LIN {X 0,Y 573.263,Z 379.078,A -85,B 0,C 180,E1 -2328.745,E2 -2328.745} C_VEL
LIN {X 0,Y 573.288,Z 379.077,A -85,B 0,C 180,E1 -2331.54,E2 -2331.54} C_VEL
LIN {X 0,Y 573.291,Z 379.075,A -85,B 0,C 180,E1 -2334.372,E2 -2334.372} C_VEL
LIN {X 0,Y 573.302,Z 379.074,A -85,B 0,C 180,E1 -2337.892,E2 -2337.892} C_VEL
LIN {X 0,Y 573.331,Z 379.07,A -85,B 0,C 180,E1 -2340.702,E2 -2340.702} C_VEL
LIN {X 0,Y 573.236,Z 379.084,A -85,B 0,C 180,E1 -2343.514,E2 -2343.514} C_VEL
LIN {X 0,Y 573.289,Z 379.075,A -85,B 0,C 180,E1 -2345.628,E2 -2345.628} C_VEL
LIN {X 0,Y 573.288,Z 379.078,A -85,B 0,C 180,E1 -2348.459,E2 -2348.459} C_VEL
LIN {X 0,Y 573.272,Z 379.077,A -85,B 0,C 180,E1 -2351.312,E2 -2351.312} C_VEL
LIN {X 0,Y 573.281,Z 379.079,A -85,B 0,C 180,E1 -2354.424,E2 -2354.424} C_VEL
LIN {X 0,Y 573.26,Z 379.079,A -85,B 0,C 180,E1 -2357.112,E2 -2357.112} C_VEL
LIN {X 0,Y 573.244,Z 379.081,A -85,B 0,C 180,E1 -2360.077,E2 -2360.077} C_VEL
LIN {X 0,Y 573.235,Z 379.082,A -85,B 0,C 180,E1 -2362.338,E2 -2362.338} C_VEL
LIN {X 0,Y 573.25,Z 379.079,A -85,B 0,C 180,E1 -2364.384,E2 -2364.384} C_VEL
LIN {X 0,Y 572.623,Z 379.16,A -85,B 0,C 180,E1 -2364.97,E2 -2364.97} C_VEL
LIN {X 0,Y 569.781,Z 379.516,A -85,B 0,C 180,E1 -2365.922,E2 -2365.922} C_VEL
LIN {X 0,Y 567.349,Z 379.82,A -85,B 0,C 180,E1 -2366.687,E2 -2366.687} C_VEL
LIN {X 0,Y 566.293,Z 379.949,A -85,B 0,C 180,E1 -2367.278,E2 -2367.278} C_VEL
LIN {X 0,Y 566.203,Z 379.958,A -85,B 0,C 180,E1 -2367.478,E2 -2367.478} C_VEL
LIN {X 0,Y 566.201,Z 379.96,A -85,B 0,C 180,E1 -2369.769,E2 -2369.769} C_VEL
LIN {X 0,Y 566.206,Z 379.959,A -85,B 0,C 180,E1 -2372.43,E2 -2372.43} C_VEL
LIN {X 0,Y 566.202,Z 379.958,A -85,B 0,C 180,E1 -2374.993,E2 -2374.993} C_VEL
LIN {X 0,Y 566.198,Z 379.957,A -85,B 0,C 180,E1 -2377.461,E2 -2377.461} C_VEL
LIN {X 0,Y 566.207,Z 379.957,A -85,B 0,C 180,E1 -2380.199,E2 -2380.199} C_VEL
LIN {X 0,Y 566.203,Z 379.96,A -85,B 0,C 180,E1 -2383.054,E2 -2383.054} C_VEL
LIN {X 0,Y 566.195,Z 379.958,A -85,B 0,C 180,E1 -2386.049,E2 -2386.049} C_VEL
LIN {X 0,Y 566.212,Z 379.959,A -85,B 0,C 180,E1 -2388.864,E2 -2388.864} C_VEL
LIN {X 0,Y 566.184,Z 379.96,A -85,B 0,C 180,E1 -2391.637,E2 -2391.637} C_VEL
LIN {X 0,Y 566.198,Z 379.958,A -85,B 0,C 180,E1 -2394.31,E2 -2394.31} C_VEL
LIN {X 0,Y 566.222,Z 379.955,A -85,B 0,C 180,E1 -2396.898,E2 -2396.898} C_VEL
LIN {X 0,Y 566.182,Z 379.961,A -85,B 0,C 180,E1 -2399.407,E2 -2399.407} C_VEL
LIN {X 0,Y 566.195,Z 379.959,A -85,B 0,C 180,E1 -2401.856,E2 -2401.856} C_VEL
LIN {X 0,Y 566.218,Z 379.957,A -85,B 0,C 180,E1 -2404.251,E2 -2404.251} C_VEL
LIN {X 0,Y 566.176,Z 379.963,A -85,B 0,C 180,E1 -2406.718,E2 -2406.718} C_VEL
LIN {X 0,Y 566.215,Z 379.956,A -85,B 0,C 180,E1 -2409.663,E2 -2409.663} C_VEL
LIN {X 0,Y 566.202,Z 379.96,A -85,B 0,C 180,E1 -2412.668,E2 -2412.668} C_VEL
LIN {X 0,Y 566.237,Z 379.953,A -85,B 0,C 180,E1 -2415.627,E2 -2415.627} C_VEL
LIN {X 0,Y 566.238,Z 379.956,A -85,B 0,C 180,E1 -2418.675,E2 -2418.675} C_VEL
LIN {X 0,Y 566.23,Z 379.955,A -85,B 0,C 180,E1 -2421.434,E2 -2421.434} C_VEL
LIN {X 0,Y 566.266,Z 379.95,A -85,B 0,C 180,E1 -2424.302,E2 -2424.302} C_VEL
LIN {X 0,Y 566.287,Z 379.947,A -85,B 0,C 180,E1 -2427.866,E2 -2427.866} C_VEL
LIN {X 0,Y 566.306,Z 379.947,A -85,B 0,C 180,E1 -2430.711,E2 -2430.711} C_VEL
LIN {X 0,Y 566.27,Z 379.95,A -85,B 0,C 180,E1 -2432.845,E2 -2432.845} C_VEL
LIN {X 0,Y 566.26,Z 379.952,A -85,B 0,C 180,E1 -2435.698,E2 -2435.698} C_VEL
LIN {X 0,Y 566.14,Z 379.968,A -85,B 0,C 180,E1 -2437.848,E2 -2437.848} C_VEL
LIN {X 0,Y 566.113,Z 380.449,A -85,B 0,C 180,E1 -2438.567,E2 -2438.567} C_VEL
LIN {X 0,Y 566.106,Z 384.738,A -85,B 0,C 180,E1 -2441.457,E2 -2441.457} C_VEL
LIN {X 0,Y 566.047,Z 389.206,A -85,B 0,C 180,E1 -2444.432,E2 -2444.432} C_VEL
LIN {X 0,Y 565.989,Z 393.668,A -85,B 0,C 180,E1 -2447.338,E2 -2447.338} C_VEL
LIN {X 0,Y 565.926,Z 397.067,A -85,B 0,C 180,E1 -2449.59,E2 -2449.59} C_VEL
LIN {X 0,Y 565.882,Z 401.918,A -85,B 0,C 180,E1 -2452.644,E2 -2452.644} C_VEL
LIN {X 0,Y 565.901,Z 405.761,A -85,B 0,C 180,E1 -2454.976,E2 -2454.976} C_VEL
LIN {X 0,Y 565.844,Z 409.742,A -85,B 0,C 180,E1 -2457.358,E2 -2457.358} C_VEL
LIN {X 0,Y 565.846,Z 414.922,A -85,B 0,C 180,E1 -2460.419,E2 -2460.419} C_VEL
LIN {X 0,Y 566.897,Z 422.356,A -85,B 0,C 180,E1 -2460.606,E2 -2460.606} C_VEL
LIN {X 0,Y 566.779,Z 435.719,A -85,B 0,C 180,E1 -2461.011,E2 -2461.011} C_VEL
LIN {X 0,Y 566.587,Z 448.306,A -85,B 0,C 180,E1 -2461.553,E2 -2461.553} C_VEL
LIN {X 0,Y 566.394,Z 460.453,A -85,B 0,C 180,E1 -2462.246,E2 -2462.246} C_VEL
LIN {X 0,Y 566.362,Z 470.852,A -85,B 0,C 180,E1 -2462.996,E2 -2462.996} C_VEL
LIN {X 0,Y 566.23,Z 480.115,A -85,B 0,C 180,E1 -2463.816,E2 -2463.816} C_VEL
LIN {X 0,Y 566.105,Z 489.376,A -85,B 0,C 180,E1 -2464.825,E2 -2464.825} C_VEL
LIN {X 0,Y 566.04,Z 497.674,A -85,B 0,C 180,E1 -2465.943,E2 -2465.943} C_VEL
LIN {X 0,Y 565.959,Z 503.812,A -85,B 0,C 180,E1 -2466.975,E2 -2466.975} C_VEL
LIN {X 0,Y 565.916,Z 508.408,A -85,B 0,C 180,E1 -2467.932,E2 -2467.932} C_VEL
LIN {X 0,Y 565.92,Z 512.057,A -85,B 0,C 180,E1 -2468.881,E2 -2468.881} C_VEL
LIN {X 0,Y 565.882,Z 515.874,A -85,B 0,C 180,E1 -2470.226,E2 -2470.226} C_VEL
LIN {X 0,Y 565.856,Z 517.602,A -85,B 0,C 180,E1 -2471.167,E2 -2471.167} C_VEL
LIN {X 0,Y 565.862,Z 518.643,A -85,B 0,C 180,E1 -2472.119,E2 -2472.119} C_VEL
LIN {X 0,Y 565.848,Z 518.997,A -85,B 0,C 180,E1 -2473.087,E2 -2473.087} C_VEL
LIN {X 0,Y 565.861,Z 518.578,A -85,B 0,C 180,E1 -2474.068,E2 -2474.068} C_VEL
LIN {X 0,Y 565.88,Z 517.38,A -85,B 0,C 180,E1 -2475.065,E2 -2475.065} C_VEL
LIN {X 0,Y 565.871,Z 515.34,A -85,B 0,C 180,E1 -2476.082,E2 -2476.082} C_VEL
LIN {X 0,Y 565.902,Z 512.383,A -85,B 0,C 180,E1 -2477.115,E2 -2477.115} C_VEL
LIN {X 0,Y 565.944,Z 508.372,A -85,B 0,C 180,E1 -2478.166,E2 -2478.166} C_VEL
LIN {X 0,Y 565.954,Z 503.101,A -85,B 0,C 180,E1 -2479.243,E2 -2479.243} C_VEL
LIN {X 0,Y 566.036,Z 496.385,A -85,B 0,C 180,E1 -2480.335,E2 -2480.335} C_VEL
LIN {X 0,Y 566.109,Z 487.815,A -85,B 0,C 180,E1 -2481.454,E2 -2481.454} C_VEL
LIN {X 0,Y 566.246,Z 478.46,A -85,B 0,C 180,E1 -2482.431,E2 -2482.431} C_VEL
LIN {X 0,Y 566.385,Z 467.752,A -85,B 0,C 180,E1 -2483.333,E2 -2483.333} C_VEL
LIN {X 0,Y 566.534,Z 457.436,A -85,B 0,C 180,E1 -2484.033,E2 -2484.033} C_VEL
LIN {X 0,Y 566.654,Z 446.742,A -85,B 0,C 180,E1 -2484.614,E2 -2484.614} C_VEL
LIN {X 0,Y 566.78,Z 434.14,A -85,B 0,C 180,E1 -2485.135,E2 -2485.135} C_VEL
LIN {X 0,Y 566.853,Z 420.783,A -85,B 0,C 180,E1 -2485.524,E2 -2485.524} C_VEL
LIN {X 0,Y 565.892,Z 414.918,A -85,B 0,C 180,E1 -2485.673,E2 -2485.673} C_VEL
LIN {X 0,Y 565.887,Z 410.031,A -85,B 0,C 180,E1 -2488.559,E2 -2488.559} C_VEL
LIN {X 0,Y 565.896,Z 405.901,A -85,B 0,C 180,E1 -2491.03,E2 -2491.03} C_VEL
LIN {X 0,Y 565.925,Z 401.919,A -85,B 0,C 180,E1 -2493.444,E2 -2493.444} C_VEL
LIN {X 0,Y 565.932,Z 398.144,A -85,B 0,C 180,E1 -2495.807,E2 -2495.807} C_VEL
LIN {X 0,Y 566.053,Z 393.562,A -85,B 0,C 180,E1 -2498.896,E2 -2498.896} C_VEL
LIN {X 0,Y 566.061,Z 390.21,A -85,B 0,C 180,E1 -2501.167,E2 -2501.167} C_VEL
LIN {X 0,Y 566.097,Z 386.758,A -85,B 0,C 180,E1 -2503.409,E2 -2503.409} C_VEL
LIN {X 0,Y 566.124,Z 382.367,A -85,B 0,C 180,E1 -2506.357,E2 -2506.357} C_VEL
LIN {X 0,Y 566.127,Z 380.228,A -85,B 0,C 180,E1 -2507.817,E2 -2507.817} C_VEL
LIN {X 0,Y 566.236,Z 379.957,A -85,B 0,C 180,E1 -2509.27,E2 -2509.27} C_VEL
LIN {X 0,Y 566.237,Z 379.955,A -85,B 0,C 180,E1 -2512.153,E2 -2512.153} C_VEL
LIN {X 0,Y 566.282,Z 379.948,A -85,B 0,C 180,E1 -2515.016,E2 -2515.016} C_VEL
LIN {X 0,Y 566.274,Z 379.95,A -85,B 0,C 180,E1 -2517.866,E2 -2517.866} C_VEL
LIN {X 0,Y 566.304,Z 379.948,A -85,B 0,C 180,E1 -2520.711,E2 -2520.711} C_VEL
LIN {X 0,Y 566.269,Z 379.952,A -85,B 0,C 180,E1 -2522.846,E2 -2522.846} C_VEL
LIN {X 0,Y 566.259,Z 379.952,A -85,B 0,C 180,E1 -2525.698,E2 -2525.698} C_VEL
LIN {X 0,Y 566.23,Z 379.955,A -85,B 0,C 180,E1 -2528.566,E2 -2528.566} C_VEL
LIN {X 0,Y 566.238,Z 379.954,A -85,B 0,C 180,E1 -2531.454,E2 -2531.454} C_VEL
LIN {X 0,Y 566.231,Z 379.955,A -85,B 0,C 180,E1 -2534.507,E2 -2534.507} C_VEL
LIN {X 0,Y 566.202,Z 379.961,A -85,B 0,C 180,E1 -2537.332,E2 -2537.332} C_VEL
LIN {X 0,Y 566.217,Z 379.958,A -85,B 0,C 180,E1 -2540.337,E2 -2540.337} C_VEL
LIN {X 0,Y 566.186,Z 379.961,A -85,B 0,C 180,E1 -2543.404,E2 -2543.404} C_VEL
LIN {X 0,Y 566.222,Z 379.958,A -85,B 0,C 180,E1 -2545.749,E2 -2545.749} C_VEL
LIN {X 0,Y 566.203,Z 379.958,A -85,B 0,C 180,E1 -2548.203,E2 -2548.203} C_VEL
LIN {X 0,Y 566.188,Z 379.961,A -85,B 0,C 180,E1 -2550.593,E2 -2550.593} C_VEL
LIN {X 0,Y 566.226,Z 379.957,A -85,B 0,C 180,E1 -2553.102,E2 -2553.102} C_VEL
LIN {X 0,Y 566.213,Z 379.959,A -85,B 0,C 180,E1 -2556.217,E2 -2556.217} C_VEL
LIN {X 0,Y 566.22,Z 379.959,A -85,B 0,C 180,E1 -2559.273,E2 -2559.273} C_VEL
LIN {X 0,Y 566.212,Z 379.958,A -85,B 0,C 180,E1 -2562.088,E2 -2562.088} C_VEL
LIN {X 0,Y 566.17,Z 379.962,A -85,B 0,C 180,E1 -2565.036,E2 -2565.036} C_VEL
LIN {X 0,Y 566.217,Z 379.956,A -85,B 0,C 180,E1 -2568.136,E2 -2568.136} C_VEL
LIN {X 0,Y 566.221,Z 379.958,A -85,B 0,C 180,E1 -2570.728,E2 -2570.728} C_VEL
LIN {X 0,Y 566.267,Z 379.999,A -85,B 0,C 180,E1 -2573.325,E2 -2573.325} C_VEL
LIN {X 0,Y 566.625,Z 384.154,A -85,B 0,C 180,E1 -2574.947,E2 -2574.947} C_VEL
LIN {X 0,Y 566.535,Z 391.153,A -85,B 0,C 180,E1 -2577.518,E2 -2577.518} C_VEL
LIN {X 0,Y 566.424,Z 399.162,A -85,B 0,C 180,E1 -2580.289,E2 -2580.289} C_VEL
LIN {X 0,Y 566.313,Z 408.642,A -85,B 0,C 180,E1 -2583.464,E2 -2583.464} C_VEL
LIN {X 0,Y 566.255,Z 417.036,A -85,B 0,C 180,E1 -2586.211,E2 -2586.211} C_VEL
LIN {X 0,Y 566.194,Z 425.345,A -85,B 0,C 180,E1 -2588.902,E2 -2588.902} C_VEL
LIN {X 0,Y 566.104,Z 433.628,A -85,B 0,C 180,E1 -2591.545,E2 -2591.545} C_VEL
LIN {X 0,Y 566.039,Z 443.095,A -85,B 0,C 180,E1 -2594.518,E2 -2594.518} C_VEL
LIN {X 0,Y 566.007,Z 452.192,A -85,B 0,C 180,E1 -2597.336,E2 -2597.336} C_VEL
LIN {X 0,Y 566.933,Z 459.527,A -85,B 0,C 180,E1 -2597.494,E2 -2597.494} C_VEL
LIN {X 0,Y 566.835,Z 471.886,A -85,B 0,C 180,E1 -2597.832,E2 -2597.832} C_VEL
LIN {X 0,Y 566.678,Z 484.291,A -85,B 0,C 180,E1 -2598.318,E2 -2598.318} C_VEL
LIN {X 0,Y 566.547,Z 496.426,A -85,B 0,C 180,E1 -2598.952,E2 -2598.952} C_VEL
LIN {X 0,Y 566.441,Z 506.751,A -85,B 0,C 180,E1 -2599.636,E2 -2599.636} C_VEL
LIN {X 0,Y 566.301,Z 515.651,A -85,B 0,C 180,E1 -2600.356,E2 -2600.356} C_VEL
LIN {X 0,Y 566.166,Z 524.79,A -85,B 0,C 180,E1 -2601.254,E2 -2601.254} C_VEL
LIN {X 0,Y 566.08,Z 533.692,A -85,B 0,C 180,E1 -2602.331,E2 -2602.331} C_VEL
LIN {X 0,Y 565.967,Z 540.958,A -85,B 0,C 180,E1 -2603.423,E2 -2603.423} C_VEL
LIN {X 0,Y 566.004,Z 545.682,A -85,B 0,C 180,E1 -2604.299,E2 -2604.299} C_VEL
LIN {X 0,Y 565.933,Z 550.373,A -85,B 0,C 180,E1 -2605.37,E2 -2605.37} C_VEL
LIN {X 0,Y 565.927,Z 553.958,A -85,B 0,C 180,E1 -2606.44,E2 -2606.44} C_VEL
LIN {X 0,Y 565.878,Z 555.809,A -85,B 0,C 180,E1 -2607.153,E2 -2607.153} C_VEL
LIN {X 0,Y 565.846,Z 558.186,A -85,B 0,C 180,E1 -2608.577,E2 -2608.577} C_VEL
LIN {X 0,Y 565.839,Z 559,A -85,B 0,C 180,E1 -2610,E2 -2610} C_VEL
LIN {X 0,Y 565.846,Z 558.186,A -85,B 0,C 180,E1 -2611.424,E2 -2611.424} C_VEL
LIN {X 0,Y 565.878,Z 555.809,A -85,B 0,C 180,E1 -2612.848,E2 -2612.848} C_VEL
LIN {X 0,Y 565.926,Z 552.895,A -85,B 0,C 180,E1 -2613.917,E2 -2613.917} C_VEL
LIN {X 0,Y 565.878,Z 548.948,A -85,B 0,C 180,E1 -2614.988,E2 -2614.988} C_VEL
LIN {X 0,Y 566.002,Z 543.866,A -85,B 0,C 180,E1 -2616.059,E2 -2616.059} C_VEL
LIN {X 0,Y 566.04,Z 537.467,A -85,B 0,C 180,E1 -2617.133,E2 -2617.133} C_VEL
LIN {X 0,Y 566.134,Z 529.476,A -85,B 0,C 180,E1 -2618.208,E2 -2618.208} C_VEL
LIN {X 0,Y 566.229,Z 521.334,A -85,B 0,C 180,E1 -2619.106,E2 -2619.106} C_VEL
LIN {X 0,Y 566.346,Z 511.398,A -85,B 0,C 180,E1 -2620.005,E2 -2620.005} C_VEL
LIN {X 0,Y 566.523,Z 500.318,A -85,B 0,C 180,E1 -2620.806,E2 -2620.806} C_VEL
LIN {X 0,Y 566.609,Z 487.943,A -85,B 0,C 180,E1 -2621.51,E2 -2621.51} C_VEL
LIN {X 0,Y 566.752,Z 475.762,A -85,B 0,C 180,E1 -2622.034,E2 -2622.034} C_VEL
LIN {X 0,Y 566.914,Z 462.34,A -85,B 0,C 180,E1 -2622.439,E2 -2622.439} C_VEL
LIN {X 0,Y 566.69,Z 456.459,A -85,B 0,C 180,E1 -2622.573,E2 -2622.573} C_VEL
LIN {X 0,Y 566.006,Z 452.19,A -85,B 0,C 180,E1 -2622.664,E2 -2622.664} C_VEL
LIN {X 0,Y 566.04,Z 443.093,A -85,B 0,C 180,E1 -2625.483,E2 -2625.483} C_VEL
LIN {X 0,Y 566.104,Z 433.626,A -85,B 0,C 180,E1 -2628.456,E2 -2628.456} C_VEL
LIN {X 0,Y 566.204,Z 424.35,A -85,B 0,C 180,E1 -2631.418,E2 -2631.418} C_VEL
LIN {X 0,Y 566.273,Z 414.636,A -85,B 0,C 180,E1 -2634.568,E2 -2634.568} C_VEL
LIN {X 0,Y 566.349,Z 406.236,A -85,B 0,C 180,E1 -2637.332,E2 -2637.332} C_VEL
LIN {X 0,Y 566.428,Z 397.82,A -85,B 0,C 180,E1 -2640.166,E2 -2640.166} C_VEL
LIN {X 0,Y 566.568,Z 389.577,A -85,B 0,C 180,E1 -2643.079,E2 -2643.079} C_VEL
LIN {X 0,Y 566.627,Z 384.22,A -85,B 0,C 180,E1 -2645.054,E2 -2645.054} C_VEL
LIN {X 0,Y 566.223,Z 379.957,A -85,B 0,C 180,E1 -2646.734,E2 -2646.734} C_VEL
LIN {X 0,Y 566.223,Z 379.957,A -85,B 0,C 180,E1 -2649.686,E2 -2649.686} C_VEL
LIN {X 0,Y 566.213,Z 379.958,A -85,B 0,C 180,E1 -2652.087,E2 -2652.087} C_VEL
LIN {X 0,Y 566.171,Z 379.962,A -85,B 0,C 180,E1 -2655.036,E2 -2655.036} C_VEL
LIN {X 0,Y 566.19,Z 379.959,A -85,B 0,C 180,E1 -2657.91,E2 -2657.91} C_VEL
LIN {X 0,Y 566.215,Z 379.959,A -85,B 0,C 180,E1 -2660.726,E2 -2660.726} C_VEL
LIN {X 0,Y 566.206,Z 379.957,A -85,B 0,C 180,E1 -2663.785,E2 -2663.785} C_VEL
LIN {X 0,Y 566.198,Z 379.958,A -85,B 0,C 180,E1 -2666.268,E2 -2666.268} C_VEL
LIN {X 0,Y 566.192,Z 379.961,A -85,B 0,C 180,E1 -2668.923,E2 -2668.923} C_VEL
LIN {X 0,Y 566.212,Z 379.956,A -85,B 0,C 180,E1 -2671.857,E2 -2671.857} C_VEL
LIN {X 0,Y 566.212,Z 379.956,A -85,B 0,C 180,E1 -2674.251,E2 -2674.251} C_VEL
LIN {X 0,Y 566.174,Z 379.961,A -85,B 0,C 180,E1 -2676.718,E2 -2676.718} C_VEL
LIN {X 0,Y 566.209,Z 379.959,A -85,B 0,C 180,E1 -2679.663,E2 -2679.663} C_VEL
LIN {X 0,Y 566.2,Z 379.958,A -85,B 0,C 180,E1 -2682.668,E2 -2682.668} C_VEL
LIN {X 0,Y 566.234,Z 379.956,A -85,B 0,C 180,E1 -2685.627,E2 -2685.627} C_VEL
LIN {X 0,Y 566.235,Z 379.953,A -85,B 0,C 180,E1 -2688.675,E2 -2688.675} C_VEL
LIN {X 0,Y 566.233,Z 379.955,A -85,B 0,C 180,E1 -2691.434,E2 -2691.434} C_VEL
LIN {X 0,Y 566.259,Z 379.952,A -85,B 0,C 180,E1 -2694.302,E2 -2694.302} C_VEL
LIN {X 0,Y 566.274,Z 379.95,A -85,B 0,C 180,E1 -2697.866,E2 -2697.866} C_VEL
LIN {X 0,Y 566.301,Z 379.945,A -85,B 0,C 180,E1 -2700.711,E2 -2700.711} C_VEL
LIN {X 0,Y 566.277,Z 379.949,A -85,B 0,C 180,E1 -2702.845,E2 -2702.845} C_VEL
LIN {X 0,Y 566.258,Z 379.951,A -85,B 0,C 180,E1 -2705.698,E2 -2705.698} C_VEL
LIN {X 0,Y 566.233,Z 379.956,A -85,B 0,C 180,E1 -2708.566,E2 -2708.566} C_VEL
LIN {X 0,Y 566.242,Z 379.952,A -85,B 0,C 180,E1 -2711.454,E2 -2711.454} C_VEL
LIN {X 0,Y 566.234,Z 379.956,A -85,B 0,C 180,E1 -2714.506,E2 -2714.506} C_VEL
LIN {X 0,Y 566.203,Z 379.957,A -85,B 0,C 180,E1 -2717.332,E2 -2717.332} C_VEL
LIN {X 0,Y 566.209,Z 379.96,A -85,B 0,C 180,E1 -2720.337,E2 -2720.337} C_VEL
LIN {X 0,Y 566.173,Z 379.961,A -85,B 0,C 180,E1 -2723.282,E2 -2723.282} C_VEL
LIN {X 0,Y 566.209,Z 379.956,A -85,B 0,C 180,E1 -2725.749,E2 -2725.749} C_VEL
LIN {X 0,Y 566.203,Z 379.958,A -85,B 0,C 180,E1 -2727.478,E2 -2727.478} C_VEL
LIN {X 0,Y 565.523,Z 380.042,A -85,B 0,C 180,E1 -2728.072,E2 -2728.072} C_VEL
LIN {X 0,Y 562.657,Z 380.399,A -85,B 0,C 180,E1 -2729.036,E2 -2729.036} C_VEL
LIN {X 0,Y 560.248,Z 380.701,A -85,B 0,C 180,E1 -2729.811,E2 -2729.811} C_VEL
LIN {X 0,Y 559.22,Z 380.827,A -85,B 0,C 180,E1 -2730.41,E2 -2730.41} C_VEL
LIN {X 0,Y 559.14,Z 380.837,A -85,B 0,C 180,E1 -2730.613,E2 -2730.613} C_VEL
LIN {X 0,Y 559.166,Z 380.836,A -85,B 0,C 180,E1 -2733.575,E2 -2733.575} C_VEL
LIN {X 0,Y 559.169,Z 380.834,A -85,B 0,C 180,E1 -2736.448,E2 -2736.448} C_VEL
LIN {X 0,Y 559.175,Z 380.833,A -85,B 0,C 180,E1 -2738.934,E2 -2738.934} C_VEL
LIN {X 0,Y 559.166,Z 380.836,A -85,B 0,C 180,E1 -2741.77,E2 -2741.77} C_VEL
LIN {X 0,Y 559.137,Z 380.838,A -85,B 0,C 180,E1 -2744.74,E2 -2744.74} C_VEL
LIN {X 0,Y 559.178,Z 380.835,A -85,B 0,C 180,E1 -2747.863,E2 -2747.863} C_VEL
LIN {X 0,Y 559.18,Z 380.835,A -85,B 0,C 180,E1 -2750.134,E2 -2750.134} C_VEL
LIN {X 0,Y 559.146,Z 380.837,A -85,B 0,C 180,E1 -2752.892,E2 -2752.892} C_VEL
LIN {X 0,Y 559.167,Z 380.836,A -85,B 0,C 180,E1 -2756.051,E2 -2756.051} C_VEL
LIN {X 0,Y 559.156,Z 380.835,A -85,B 0,C 180,E1 -2758.981,E2 -2758.981} C_VEL
LIN {X 0,Y 559.17,Z 380.833,A -85,B 0,C 180,E1 -2761.619,E2 -2761.619} C_VEL
LIN {X 0,Y 559.184,Z 380.831,A -85,B 0,C 180,E1 -2763.903,E2 -2763.903} C_VEL
LIN {X 0,Y 559.145,Z 380.838,A -85,B 0,C 180,E1 -2766.571,E2 -2766.571} C_VEL
LIN {X 0,Y 559.181,Z 380.834,A -85,B 0,C 180,E1 -2769.395,E2 -2769.395} C_VEL
LIN {X 0,Y 559.145,Z 380.839,A -85,B 0,C 180,E1 -2771.686,E2 -2771.686} C_VEL
LIN {X 0,Y 559.163,Z 380.836,A -85,B 0,C 180,E1 -2773.948,E2 -2773.948} C_VEL
LIN {X 0,Y 559.173,Z 380.834,A -85,B 0,C 180,E1 -2776.184,E2 -2776.184} C_VEL
LIN {X 0,Y 559.209,Z 380.831,A -85,B 0,C 180,E1 -2778.605,E2 -2778.605} C_VEL
LIN {X 0,Y 559.202,Z 380.83,A -85,B 0,C 180,E1 -2782.053,E2 -2782.053} C_VEL
LIN {X 0,Y 559.252,Z 380.824,A -85,B 0,C 180,E1 -2784.953,E2 -2784.953} C_VEL
LIN {X 0,Y 559.257,Z 380.822,A -85,B 0,C 180,E1 -2787.839,E2 -2787.839} C_VEL
LIN {X 0,Y 559.276,Z 380.823,A -85,B 0,C 180,E1 -2790.72,E2 -2790.72} C_VEL
LIN {X 0,Y 559.237,Z 380.827,A -85,B 0,C 180,E1 -2792.881,E2 -2792.881} C_VEL
LIN {X 0,Y 559.228,Z 380.827,A -85,B 0,C 180,E1 -2795.77,E2 -2795.77} C_VEL
LIN {X 0,Y 559.097,Z 380.846,A -85,B 0,C 180,E1 -2797.948,E2 -2797.948} C_VEL
LIN {X 0,Y 559.052,Z 381.385,A -85,B 0,C 180,E1 -2798.676,E2 -2798.676} C_VEL
LIN {X 0,Y 559.024,Z 385.689,A -85,B 0,C 180,E1 -2801.604,E2 -2801.604} C_VEL
LIN {X 0,Y 558.962,Z 390.082,A -85,B 0,C 180,E1 -2804.564,E2 -2804.564} C_VEL
LIN {X 0,Y 558.914,Z 394.671,A -85,B 0,C 180,E1 -2807.564,E2 -2807.564} C_VEL
LIN {X 0,Y 558.846,Z 398.083,A -85,B 0,C 180,E1 -2809.849,E2 -2809.849} C_VEL
LIN {X 0,Y 558.809,Z 402.844,A -85,B 0,C 180,E1 -2812.947,E2 -2812.947} C_VEL
LIN {X 0,Y 558.811,Z 406.706,A -85,B 0,C 180,E1 -2815.315,E2 -2815.315} C_VEL
LIN {X 0,Y 558.733,Z 411.646,A -85,B 0,C 180,E1 -2818.298,E2 -2818.298} C_VEL
LIN {X 0,Y 558.768,Z 414.924,A -85,B 0,C 180,E1 -2820.257,E2 -2820.257} C_VEL
LIN {X 0,Y 559.968,Z 423.248,A -85,B 0,C 180,E1 -2820.472,E2 -2820.472} C_VEL
LIN {X 0,Y 559.822,Z 436.116,A -85,B 0,C 180,E1 -2820.873,E2 -2820.873} C_VEL
LIN {X 0,Y 559.619,Z 448.317,A -85,B 0,C 180,E1 -2821.409,E2 -2821.409} C_VEL
LIN {X 0,Y 559.435,Z 459.64,A -85,B 0,C 180,E1 -2822.057,E2 -2822.057} C_VEL
LIN {X 0,Y 559.323,Z 470.12,A -85,B 0,C 180,E1 -2822.811,E2 -2822.811} C_VEL
LIN {X 0,Y 559.206,Z 478.794,A -85,B 0,C 180,E1 -2823.571,E2 -2823.571} C_VEL
LIN {X 0,Y 559.113,Z 487.101,A -85,B 0,C 180,E1 -2824.446,E2 -2824.446} C_VEL
LIN {X 0,Y 558.972,Z 495.662,A -85,B 0,C 180,E1 -2825.556,E2 -2825.556} C_VEL
LIN {X 0,Y 558.903,Z 502.976,A -85,B 0,C 180,E1 -2826.746,E2 -2826.746} C_VEL
LIN {X 0,Y 558.833,Z 507.214,A -85,B 0,C 180,E1 -2827.599,E2 -2827.599} C_VEL
LIN {X 0,Y 558.826,Z 511.836,A -85,B 0,C 180,E1 -2828.764,E2 -2828.764} C_VEL
LIN {X 0,Y 558.8,Z 515.166,A -85,B 0,C 180,E1 -2829.897,E2 -2829.897} C_VEL
LIN {X 0,Y 558.748,Z 517.384,A -85,B 0,C 180,E1 -2831.002,E2 -2831.002} C_VEL
LIN {X 0,Y 558.762,Z 518.632,A -85,B 0,C 180,E1 -2832.09,E2 -2832.09} C_VEL
LIN {X 0,Y 558.761,Z 518.983,A -85,B 0,C 180,E1 -2833.154,E2 -2833.154} C_VEL
LIN {X 0,Y 558.778,Z 518.492,A -85,B 0,C 180,E1 -2834.2,E2 -2834.2} C_VEL
LIN {X 0,Y 558.791,Z 517.169,A -85,B 0,C 180,E1 -2835.225,E2 -2835.225} C_VEL
LIN {X 0,Y 558.784,Z 515.069,A -85,B 0,C 180,E1 -2836.231,E2 -2836.231} C_VEL
LIN {X 0,Y 558.835,Z 510.936,A -85,B 0,C 180,E1 -2837.588,E2 -2837.588} C_VEL
LIN {X 0,Y 558.872,Z 506.636,A -85,B 0,C 180,E1 -2838.621,E2 -2838.621} C_VEL
LIN {X 0,Y 558.918,Z 499.913,A -85,B 0,C 180,E1 -2839.877,E2 -2839.877} C_VEL
LIN {X 0,Y 559.028,Z 491.888,A -85,B 0,C 180,E1 -2841.054,E2 -2841.054} C_VEL
LIN {X 0,Y 559.168,Z 483.036,A -85,B 0,C 180,E1 -2842.092,E2 -2842.092} C_VEL
LIN {X 0,Y 559.326,Z 472.596,A -85,B 0,C 180,E1 -2843.075,E2 -2843.075} C_VEL
LIN {X 0,Y 559.496,Z 462.88,A -85,B 0,C 180,E1 -2843.816,E2 -2843.816} C_VEL
LIN {X 0,Y 559.628,Z 451.149,A -85,B 0,C 180,E1 -2844.533,E2 -2844.533} C_VEL
LIN {X 0,Y 559.814,Z 438.793,A -85,B 0,C 180,E1 -2845.11,E2 -2845.11} C_VEL
LIN {X 0,Y 559.915,Z 425.764,A -85,B 0,C 180,E1 -2845.555,E2 -2845.555} C_VEL
LIN {X 0,Y 559.789,Z 420.982,A -85,B 0,C 180,E1 -2845.679,E2 -2845.679} C_VEL
LIN {X 0,Y 558.793,Z 414.9,A -85,B 0,C 180,E1 -2845.846,E2 -2845.846} C_VEL
LIN {X 0,Y 558.781,Z 409.706,A -85,B 0,C 180,E1 -2848.958,E2 -2848.958} C_VEL
LIN {X 0,Y 558.84,Z 405.222,A -85,B 0,C 180,E1 -2851.68,E2 -2851.68} C_VEL
LIN {X 0,Y 558.843,Z 400.485,A -85,B 0,C 180,E1 -2854.686,E2 -2854.686} C_VEL
LIN {X 0,Y 558.896,Z 396.959,A -85,B 0,C 180,E1 -2857.057,E2 -2857.057} C_VEL
LIN {X 0,Y 558.975,Z 393.58,A -85,B 0,C 180,E1 -2859.388,E2 -2859.388} C_VEL
LIN {X 0,Y 558.977,Z 390.097,A -85,B 0,C 180,E1 -2861.68,E2 -2861.68} C_VEL
LIN {X 0,Y 559.018,Z 386.686,A -85,B 0,C 180,E1 -2863.944,E2 -2863.944} C_VEL
LIN {X 0,Y 559.057,Z 383.42,A -85,B 0,C 180,E1 -2866.181,E2 -2866.181} C_VEL
LIN {X 0,Y 559.073,Z 381.267,A -85,B 0,C 180,E1 -2867.661,E2 -2867.661} C_VEL
LIN {X 0,Y 559.151,Z 380.837,A -85,B 0,C 180,E1 -2868.63,E2 -2868.63} C_VEL
LIN {X 0,Y 559.199,Z 380.834,A -85,B 0,C 180,E1 -2871.326,E2 -2871.326} C_VEL
LIN {X 0,Y 559.225,Z 380.828,A -85,B 0,C 180,E1 -2874.23,E2 -2874.23} C_VEL
LIN {X 0,Y 559.241,Z 380.826,A -85,B 0,C 180,E1 -2877.119,E2 -2877.119} C_VEL
LIN {X 0,Y 559.256,Z 380.824,A -85,B 0,C 180,E1 -2880,E2 -2880} C_VEL
LIN {X 0,Y 559.236,Z 380.828,A -85,B 0,C 180,E1 -2882.881,E2 -2882.881} C_VEL
LIN {X 0,Y 559.228,Z 380.828,A -85,B 0,C 180,E1 -2885.77,E2 -2885.77} C_VEL
LIN {X 0,Y 559.188,Z 380.832,A -85,B 0,C 180,E1 -2888.674,E2 -2888.674} C_VEL
LIN {X 0,Y 559.201,Z 380.83,A -85,B 0,C 180,E1 -2891.601,E2 -2891.601} C_VEL
LIN {X 0,Y 559.195,Z 380.831,A -85,B 0,C 180,E1 -2894.596,E2 -2894.596} C_VEL
LIN {X 0,Y 559.161,Z 380.836,A -85,B 0,C 180,E1 -2897.557,E2 -2897.557} C_VEL
LIN {X 0,Y 559.172,Z 380.834,A -85,B 0,C 180,E1 -2899.837,E2 -2899.837} C_VEL
LIN {X 0,Y 559.139,Z 380.838,A -85,B 0,C 180,E1 -2902.153,E2 -2902.153} C_VEL
LIN {X 0,Y 559.176,Z 380.833,A -85,B 0,C 180,E1 -2905.188,E2 -2905.188} C_VEL
LIN {X 0,Y 559.192,Z 380.834,A -85,B 0,C 180,E1 -2907.712,E2 -2907.712} C_VEL
LIN {X 0,Y 559.164,Z 380.835,A -85,B 0,C 180,E1 -2910.182,E2 -2910.182} C_VEL
LIN {X 0,Y 559.172,Z 380.835,A -85,B 0,C 180,E1 -2912.714,E2 -2912.714} C_VEL
LIN {X 0,Y 559.147,Z 380.838,A -85,B 0,C 180,E1 -2915.323,E2 -2915.323} C_VEL
LIN {X 0,Y 559.134,Z 380.841,A -85,B 0,C 180,E1 -2918.018,E2 -2918.018} C_VEL
LIN {X 0,Y 559.175,Z 380.834,A -85,B 0,C 180,E1 -2920.811,E2 -2920.811} C_VEL
LIN {X 0,Y 559.14,Z 380.839,A -85,B 0,C 180,E1 -2923.734,E2 -2923.734} C_VEL
LIN {X 0,Y 559.143,Z 380.838,A -85,B 0,C 180,E1 -2926.804,E2 -2926.804} C_VEL
LIN {X 0,Y 559.176,Z 380.834,A -85,B 0,C 180,E1 -2929.19,E2 -2929.19} C_VEL
LIN {X 0,Y 559.135,Z 380.84,A -85,B 0,C 180,E1 -2931.983,E2 -2931.983} C_VEL
LIN {X 0,Y 559.201,Z 380.946,A -85,B 0,C 180,E1 -2933.156,E2 -2933.156} C_VEL
LIN {X 0,Y 559.641,Z 384.806,A -85,B 0,C 180,E1 -2934.714,E2 -2934.714} C_VEL
LIN {X 0,Y 559.542,Z 391.763,A -85,B 0,C 180,E1 -2937.311,E2 -2937.311} C_VEL
LIN {X 0,Y 559.404,Z 399.619,A -85,B 0,C 180,E1 -2940.098,E2 -2940.098} C_VEL
LIN {X 0,Y 559.281,Z 408.63,A -85,B 0,C 180,E1 -2943.151,E2 -2943.151} C_VEL
LIN {X 0,Y 559.216,Z 416.889,A -85,B 0,C 180,E1 -2945.893,E2 -2945.893} C_VEL
LIN {X 0,Y 559.147,Z 425.344,A -85,B 0,C 180,E1 -2948.623,E2 -2948.623} C_VEL
LIN {X 0,Y 559.055,Z 434.811,A -85,B 0,C 180,E1 -2951.683,E2 -2951.683} C_VEL
LIN {X 0,Y 558.983,Z 444.278,A -85,B 0,C 180,E1 -2954.691,E2 -2954.691} C_VEL
LIN {X 0,Y 558.928,Z 452.192,A -85,B 0,C 180,E1 -2957.173,E2 -2957.173} C_VEL
LIN {X 0,Y 560.011,Z 459.527,A -85,B 0,C 180,E1 -2957.337,E2 -2957.337} C_VEL
LIN {X 0,Y 559.898,Z 471.886,A -85,B 0,C 180,E1 -2957.679,E2 -2957.679} C_VEL
LIN {X 0,Y 559.722,Z 484.289,A -85,B 0,C 180,E1 -2958.171,E2 -2958.171} C_VEL
LIN {X 0,Y 559.552,Z 495.711,A -85,B 0,C 180,E1 -2958.77,E2 -2958.77} C_VEL
LIN {X 0,Y 559.428,Z 506.75,A -85,B 0,C 180,E1 -2959.505,E2 -2959.505} C_VEL
LIN {X 0,Y 559.244,Z 517.604,A -85,B 0,C 180,E1 -2960.415,E2 -2960.415} C_VEL
LIN {X 0,Y 559.127,Z 526.416,A -85,B 0,C 180,E1 -2961.325,E2 -2961.325} C_VEL
LIN {X 0,Y 558.996,Z 535.004,A -85,B 0,C 180,E1 -2962.414,E2 -2962.414} C_VEL
LIN {X 0,Y 558.885,Z 542.686,A -85,B 0,C 180,E1 -2963.649,E2 -2963.649} C_VEL
LIN {X 0,Y 558.869,Z 547.367,A -85,B 0,C 180,E1 -2964.588,E2 -2964.588} C_VEL
LIN {X 0,Y 558.869,Z 551.678,A -85,B 0,C 180,E1 -2965.673,E2 -2965.673} C_VEL
LIN {X 0,Y 558.836,Z 553.958,A -85,B 0,C 180,E1 -2966.395,E2 -2966.395} C_VEL
LIN {X 0,Y 558.799,Z 555.809,A -85,B 0,C 180,E1 -2967.117,E2 -2967.117} C_VEL
LIN {X 0,Y 558.745,Z 558.185,A -85,B 0,C 180,E1 -2968.559,E2 -2968.559} C_VEL
LIN {X 0,Y 558.74,Z 559,A -85,B 0,C 180,E1 -2970,E2 -2970} C_VEL
LIN {X 0,Y 558.745,Z 558.185,A -85,B 0,C 180,E1 -2971.442,E2 -2971.442} C_VEL
LIN {X 0,Y 558.799,Z 555.809,A -85,B 0,C 180,E1 -2972.884,E2 -2972.884} C_VEL
LIN {X 0,Y 558.844,Z 552.895,A -85,B 0,C 180,E1 -2973.966,E2 -2973.966} C_VEL
LIN {X 0,Y 558.798,Z 548.948,A -85,B 0,C 180,E1 -2975.051,E2 -2975.051} C_VEL
LIN {X 0,Y 558.921,Z 543.866,A -85,B 0,C 180,E1 -2976.136,E2 -2976.136} C_VEL
LIN {X 0,Y 558.977,Z 537.466,A -85,B 0,C 180,E1 -2977.223,E2 -2977.223} C_VEL
LIN {X 0,Y 559.099,Z 529.476,A -85,B 0,C 180,E1 -2978.312,E2 -2978.312} C_VEL
LIN {X 0,Y 559.195,Z 521.333,A -85,B 0,C 180,E1 -2979.221,E2 -2979.221} C_VEL
LIN {X 0,Y 559.347,Z 511.398,A -85,B 0,C 180,E1 -2980.132,E2 -2980.132} C_VEL
LIN {X 0,Y 559.539,Z 500.424,A -85,B 0,C 180,E1 -2980.935,E2 -2980.935} C_VEL
LIN {X 0,Y 559.636,Z 488.815,A -85,B 0,C 180,E1 -2981.61,E2 -2981.61} C_VEL
LIN {X 0,Y 559.798,Z 476.977,A -85,B 0,C 180,E1 -2982.139,E2 -2982.139} C_VEL
LIN {X 0,Y 559.971,Z 464.168,A -85,B 0,C 180,E1 -2982.55,E2 -2982.55} C_VEL
LIN {X 0,Y 559.865,Z 457.941,A -85,B 0,C 180,E1 -2982.699,E2 -2982.699} C_VEL
LIN {X 0,Y 558.927,Z 452.19,A -85,B 0,C 180,E1 -2982.827,E2 -2982.827} C_VEL
LIN {X 0,Y 558.976,Z 443.093,A -85,B 0,C 180,E1 -2985.683,E2 -2985.683} C_VEL
LIN {X 0,Y 559.073,Z 433.626,A -85,B 0,C 180,E1 -2988.697,E2 -2988.697} C_VEL
LIN {X 0,Y 559.153,Z 424.808,A -85,B 0,C 180,E1 -2991.548,E2 -2991.548} C_VEL
LIN {X 0,Y 559.22,Z 415.759,A -85,B 0,C 180,E1 -2994.502,E2 -2994.502} C_VEL
LIN {X 0,Y 559.334,Z 407.359,A -85,B 0,C 180,E1 -2997.298,E2 -2997.298} C_VEL
LIN {X 0,Y 559.417,Z 398.943,A -85,B 0,C 180,E1 -3000.167,E2 -3000.167} C_VEL
LIN {X 0,Y 559.575,Z 390.723,A -85,B 0,C 180,E1 -3003.116,E2 -3003.116} C_VEL
LIN {X 0,Y 559.644,Z 384.919,A -85,B 0,C 180,E1 -3005.287,E2 -3005.287} C_VEL
LIN {X 0,Y 559.178,Z 380.835,A -85,B 0,C 180,E1 -3006.931,E2 -3006.931} C_VEL
LIN {X 0,Y 559.167,Z 380.837,A -85,B 0,C 180,E1 -3009.942,E2 -3009.942} C_VEL
LIN {X 0,Y 559.162,Z 380.835,A -85,B 0,C 180,E1 -3012.743,E2 -3012.743} C_VEL
LIN {X 0,Y 559.153,Z 380.838,A -85,B 0,C 180,E1 -3015.761,E2 -3015.761} C_VEL
LIN {X 0,Y 559.164,Z 380.837,A -85,B 0,C 180,E1 -3018.23,E2 -3018.23} C_VEL
LIN {X 0,Y 559.176,Z 380.833,A -85,B 0,C 180,E1 -3021.192,E2 -3021.192} C_VEL
LIN {X 0,Y 559.161,Z 380.835,A -85,B 0,C 180,E1 -3023.791,E2 -3023.791} C_VEL
LIN {X 0,Y 559.149,Z 380.837,A -85,B 0,C 180,E1 -3026.424,E2 -3026.424} C_VEL
LIN {X 0,Y 559.156,Z 380.838,A -85,B 0,C 180,E1 -3028.981,E2 -3028.981} C_VEL
LIN {X 0,Y 559.169,Z 380.834,A -85,B 0,C 180,E1 -3031.619,E2 -3031.619} C_VEL
LIN {X 0,Y 559.18,Z 380.834,A -85,B 0,C 180,E1 -3033.903,E2 -3033.903} C_VEL
LIN {X 0,Y 559.143,Z 380.837,A -85,B 0,C 180,E1 -3036.571,E2 -3036.571} C_VEL
LIN {X 0,Y 559.178,Z 380.833,A -85,B 0,C 180,E1 -3039.395,E2 -3039.395} C_VEL
LIN {X 0,Y 559.143,Z 380.837,A -85,B 0,C 180,E1 -3041.686,E2 -3041.686} C_VEL
LIN {X 0,Y 559.165,Z 380.833,A -85,B 0,C 180,E1 -3043.948,E2 -3043.948} C_VEL
LIN {X 0,Y 559.171,Z 380.833,A -85,B 0,C 180,E1 -3046.184,E2 -3046.184} C_VEL
LIN {X 0,Y 559.194,Z 380.832,A -85,B 0,C 180,E1 -3049.133,E2 -3049.133} C_VEL
LIN {X 0,Y 559.205,Z 380.829,A -85,B 0,C 180,E1 -3052.054,E2 -3052.054} C_VEL
LIN {X 0,Y 559.254,Z 380.824,A -85,B 0,C 180,E1 -3054.953,E2 -3054.953} C_VEL
LIN {X 0,Y 559.246,Z 380.825,A -85,B 0,C 180,E1 -3057.839,E2 -3057.839} C_VEL
LIN {X 0,Y 559.272,Z 380.821,A -85,B 0,C 180,E1 -3060.72,E2 -3060.72} C_VEL
LIN {X 0,Y 559.243,Z 380.825,A -85,B 0,C 180,E1 -3062.881,E2 -3062.881} C_VEL
LIN {X 0,Y 559.228,Z 380.827,A -85,B 0,C 180,E1 -3065.77,E2 -3065.77} C_VEL
LIN {X 0,Y 559.191,Z 380.832,A -85,B 0,C 180,E1 -3068.674,E2 -3068.674} C_VEL
LIN {X 0,Y 559.205,Z 380.829,A -85,B 0,C 180,E1 -3071.6,E2 -3071.6} C_VEL
LIN {X 0,Y 559.2,Z 380.831,A -85,B 0,C 180,E1 -3074.596,E2 -3074.596} C_VEL
LIN {X 0,Y 559.163,Z 380.835,A -85,B 0,C 180,E1 -3077.557,E2 -3077.557} C_VEL
LIN {X 0,Y 559.167,Z 380.833,A -85,B 0,C 180,E1 -3079.838,E2 -3079.838} C_VEL
LIN {X 0,Y 559.141,Z 380.837,A -85,B 0,C 180,E1 -3082.153,E2 -3082.153} C_VEL
LIN {X 0,Y 559.175,Z 380.834,A -85,B 0,C 180,E1 -3085.298,E2 -3085.298} C_VEL
LIN {X 0,Y 559.181,Z 380.833,A -85,B 0,C 180,E1 -3087.712,E2 -3087.712} C_VEL
LIN {X 0,Y 559.14,Z 380.837,A -85,B 0,C 180,E1 -3090.613,E2 -3090.613} C_VEL
LIN {X 0,Y 558.48,Z 380.922,A -85,B 0,C 180,E1 -3091.214,E2 -3091.214} C_VEL
LIN {X 0,Y 555.621,Z 381.277,A -85,B 0,C 180,E1 -3092.191,E2 -3092.191} C_VEL
LIN {X 0,Y 553.21,Z 381.576,A -85,B 0,C 180,E1 -3092.976,E2 -3092.976} C_VEL
LIN {X 0,Y 552.189,Z 381.705,A -85,B 0,C 180,E1 -3093.583,E2 -3093.583} C_VEL
LIN {X 0,Y 552.114,Z 381.711,A -85,B 0,C 180,E1 -3093.788,E2 -3093.788} C_VEL
LIN {X 0,Y 552.113,Z 381.714,A -85,B 0,C 180,E1 -3096.747,E2 -3096.747} C_VEL
LIN {X 0,Y 552.13,Z 381.712,A -85,B 0,C 180,E1 -3099.527,E2 -3099.527} C_VEL
LIN {X 0,Y 552.13,Z 381.71,A -85,B 0,C 180,E1 -3102.426,E2 -3102.426} C_VEL
LIN {X 0,Y 552.094,Z 381.716,A -85,B 0,C 180,E1 -3105.562,E2 -3105.562} C_VEL
LIN {X 0,Y 552.139,Z 381.71,A -85,B 0,C 180,E1 -3108.676,E2 -3108.676} C_VEL
LIN {X 0,Y 552.117,Z 381.714,A -85,B 0,C 180,E1 -3111.411,E2 -3111.411} C_VEL
LIN {X 0,Y 552.104,Z 381.714,A -85,B 0,C 180,E1 -3114.158,E2 -3114.158} C_VEL
LIN {X 0,Y 552.117,Z 381.712,A -85,B 0,C 180,E1 -3116.814,E2 -3116.814} C_VEL
LIN {X 0,Y 552.104,Z 381.714,A -85,B 0,C 180,E1 -3119.391,E2 -3119.391} C_VEL
LIN {X 0,Y 552.107,Z 381.714,A -85,B 0,C 180,E1 -3121.901,E2 -3121.901} C_VEL
LIN {X 0,Y 552.159,Z 381.708,A -85,B 0,C 180,E1 -3124.65,E2 -3124.65} C_VEL
LIN {X 0,Y 552.094,Z 381.714,A -85,B 0,C 180,E1 -3127.549,E2 -3127.549} C_VEL
LIN {X 0,Y 552.148,Z 381.711,A -85,B 0,C 180,E1 -3130.374,E2 -3130.374} C_VEL
LIN {X 0,Y 552.136,Z 381.711,A -85,B 0,C 180,E1 -3132.977,E2 -3132.977} C_VEL
LIN {X 0,Y 552.137,Z 381.71,A -85,B 0,C 180,E1 -3136.004,E2 -3136.004} C_VEL
LIN {X 0,Y 552.164,Z 381.707,A -85,B 0,C 180,E1 -3138.993,E2 -3138.993} C_VEL
LIN {X 0,Y 552.158,Z 381.707,A -85,B 0,C 180,E1 -3141.951,E2 -3141.951} C_VEL
LIN {X 0,Y 552.228,Z 381.699,A -85,B 0,C 180,E1 -3144.889,E2 -3144.889} C_VEL
LIN {X 0,Y 552.228,Z 381.698,A -85,B 0,C 180,E1 -3147.812,E2 -3147.812} C_VEL
LIN {X 0,Y 552.246,Z 381.698,A -85,B 0,C 180,E1 -3150.729,E2 -3150.729} C_VEL
LIN {X 0,Y 552.205,Z 381.703,A -85,B 0,C 180,E1 -3152.918,E2 -3152.918} C_VEL
LIN {X 0,Y 552.198,Z 381.703,A -85,B 0,C 180,E1 -3155.844,E2 -3155.844} C_VEL
LIN {X 0,Y 552.042,Z 381.724,A -85,B 0,C 180,E1 -3158.05,E2 -3158.05} C_VEL
LIN {X 0,Y 552.001,Z 382.314,A -85,B 0,C 180,E1 -3158.788,E2 -3158.788} C_VEL
LIN {X 0,Y 551.97,Z 386.637,A -85,B 0,C 180,E1 -3161.754,E2 -3161.754} C_VEL
LIN {X 0,Y 551.875,Z 391.066,A -85,B 0,C 180,E1 -3164.755,E2 -3164.755} C_VEL
LIN {X 0,Y 551.828,Z 395.639,A -85,B 0,C 180,E1 -3167.797,E2 -3167.797} C_VEL
LIN {X 0,Y 551.755,Z 399.103,A -85,B 0,C 180,E1 -3170.115,E2 -3170.115} C_VEL
LIN {X 0,Y 551.726,Z 403.869,A -85,B 0,C 180,E1 -3173.258,E2 -3173.258} C_VEL
LIN {X 0,Y 551.698,Z 407.657,A -85,B 0,C 180,E1 -3175.665,E2 -3175.665} C_VEL
LIN {X 0,Y 551.643,Z 412.247,A -85,B 0,C 180,E1 -3178.47,E2 -3178.47} C_VEL
LIN {X 0,Y 551.69,Z 414.897,A -85,B 0,C 180,E1 -3180.074,E2 -3180.074} C_VEL
LIN {X 0,Y 553.032,Z 423.808,A -85,B 0,C 180,E1 -3180.326,E2 -3180.326} C_VEL
LIN {X 0,Y 552.893,Z 436.14,A -85,B 0,C 180,E1 -3180.719,E2 -3180.719} C_VEL
LIN {X 0,Y 552.65,Z 448.417,A -85,B 0,C 180,E1 -3181.265,E2 -3181.265} C_VEL
LIN {X 0,Y 552.442,Z 460.807,A -85,B 0,C 180,E1 -3181.992,E2 -3181.992} C_VEL
LIN {X 0,Y 552.322,Z 471.659,A -85,B 0,C 180,E1 -3182.806,E2 -3182.806} C_VEL
LIN {X 0,Y 552.157,Z 481.558,A -85,B 0,C 180,E1 -3183.729,E2 -3183.729} C_VEL
LIN {X 0,Y 551.994,Z 490.425,A -85,B 0,C 180,E1 -3184.743,E2 -3184.743} C_VEL
LIN {X 0,Y 551.887,Z 498.288,A -85,B 0,C 180,E1 -3185.858,E2 -3185.858} C_VEL
LIN {X 0,Y 551.782,Z 504.708,A -85,B 0,C 180,E1 -3187,E2 -3187} C_VEL
LIN {X 0,Y 551.753,Z 510.005,A -85,B 0,C 180,E1 -3188.201,E2 -3188.201} C_VEL
LIN {X 0,Y 551.692,Z 514.446,A -85,B 0,C 180,E1 -3189.564,E2 -3189.564} C_VEL
LIN {X 0,Y 551.676,Z 516.601,A -85,B 0,C 180,E1 -3190.519,E2 -3190.519} C_VEL
LIN {X 0,Y 551.668,Z 518.077,A -85,B 0,C 180,E1 -3191.487,E2 -3191.487} C_VEL
LIN {X 0,Y 551.652,Z 518.877,A -85,B 0,C 180,E1 -3192.47,E2 -3192.47} C_VEL
LIN {X 0,Y 551.667,Z 518.915,A -85,B 0,C 180,E1 -3193.466,E2 -3193.466} C_VEL
LIN {X 0,Y 551.701,Z 518.2,A -85,B 0,C 180,E1 -3194.49,E2 -3194.49} C_VEL
LIN {X 0,Y 551.702,Z 516.694,A -85,B 0,C 180,E1 -3195.522,E2 -3195.522} C_VEL
LIN {X 0,Y 551.688,Z 514.347,A -85,B 0,C 180,E1 -3196.562,E2 -3196.562} C_VEL
LIN {X 0,Y 551.751,Z 511.003,A -85,B 0,C 180,E1 -3197.627,E2 -3197.627} C_VEL
LIN {X 0,Y 551.795,Z 506.531,A -85,B 0,C 180,E1 -3198.716,E2 -3198.716} C_VEL
LIN {X 0,Y 551.834,Z 500.734,A -85,B 0,C 180,E1 -3199.83,E2 -3199.83} C_VEL
LIN {X 0,Y 551.957,Z 493.345,A -85,B 0,C 180,E1 -3200.959,E2 -3200.959} C_VEL
LIN {X 0,Y 552.105,Z 485.095,A -85,B 0,C 180,E1 -3201.981,E2 -3201.981} C_VEL
LIN {X 0,Y 552.252,Z 475.811,A -85,B 0,C 180,E1 -3202.922,E2 -3202.922} C_VEL
LIN {X 0,Y 552.393,Z 466.038,A -85,B 0,C 180,E1 -3203.728,E2 -3203.728} C_VEL
LIN {X 0,Y 552.59,Z 454.593,A -85,B 0,C 180,E1 -3204.485,E2 -3204.485} C_VEL
LIN {X 0,Y 552.749,Z 442.714,A -85,B 0,C 180,E1 -3205.099,E2 -3205.099} C_VEL
LIN {X 0,Y 552.972,Z 429.737,A -85,B 0,C 180,E1 -3205.593,E2 -3205.593} C_VEL
LIN {X 0,Y 552.933,Z 422.37,A -85,B 0,C 180,E1 -3205.803,E2 -3205.803} C_VEL
LIN {X 0,Y 551.7,Z 414.892,A -85,B 0,C 180,E1 -3206.019,E2 -3206.019} C_VEL
LIN {X 0,Y 551.722,Z 410.651,A -85,B 0,C 180,E1 -3208.589,E2 -3208.589} C_VEL
LIN {X 0,Y 551.748,Z 405.35,A -85,B 0,C 180,E1 -3211.882,E2 -3211.882} C_VEL
LIN {X 0,Y 551.797,Z 401.063,A -85,B 0,C 180,E1 -3214.727,E2 -3214.727} C_VEL
LIN {X 0,Y 551.832,Z 396.95,A -85,B 0,C 180,E1 -3217.538,E2 -3217.538} C_VEL
LIN {X 0,Y 551.939,Z 392.67,A -85,B 0,C 180,E1 -3220.433,E2 -3220.433} C_VEL
LIN {X 0,Y 551.956,Z 388.852,A -85,B 0,C 180,E1 -3222.971,E2 -3222.971} C_VEL
LIN {X 0,Y 552.007,Z 384.491,A -85,B 0,C 180,E1 -3226.001,E2 -3226.001} C_VEL
LIN {X 0,Y 552.011,Z 382.314,A -85,B 0,C 180,E1 -3227.5,E2 -3227.5} C_VEL
LIN {X 0,Y 552.112,Z 381.714,A -85,B 0,C 180,E1 -3228.563,E2 -3228.563} C_VEL
LIN {X 0,Y 552.167,Z 381.709,A -85,B 0,C 180,E1 -3231.214,E2 -3231.214} C_VEL
LIN {X 0,Y 552.195,Z 381.703,A -85,B 0,C 180,E1 -3234.156,E2 -3234.156} C_VEL
LIN {X 0,Y 552.207,Z 381.702,A -85,B 0,C 180,E1 -3237.082,E2 -3237.082} C_VEL
LIN {X 0,Y 552.226,Z 381.7,A -85,B 0,C 180,E1 -3240,E2 -3240} C_VEL
LIN {X 0,Y 552.202,Z 381.704,A -85,B 0,C 180,E1 -3242.918,E2 -3242.918} C_VEL
LIN {X 0,Y 552.199,Z 381.705,A -85,B 0,C 180,E1 -3245.844,E2 -3245.844} C_VEL
LIN {X 0,Y 552.159,Z 381.708,A -85,B 0,C 180,E1 -3248.786,E2 -3248.786} C_VEL
LIN {X 0,Y 552.159,Z 381.708,A -85,B 0,C 180,E1 -3251.751,E2 -3251.751} C_VEL
LIN {X 0,Y 552.133,Z 381.711,A -85,B 0,C 180,E1 -3254.749,E2 -3254.749} C_VEL
LIN {X 0,Y 552.112,Z 381.713,A -85,B 0,C 180,E1 -3257.789,E2 -3257.789} C_VEL
LIN {X 0,Y 552.131,Z 381.711,A -85,B 0,C 180,E1 -3260.101,E2 -3260.101} C_VEL
LIN {X 0,Y 552.093,Z 381.717,A -85,B 0,C 180,E1 -3262.451,E2 -3262.451} C_VEL
LIN {X 0,Y 552.154,Z 381.708,A -85,B 0,C 180,E1 -3265.351,E2 -3265.351} C_VEL
LIN {X 0,Y 552.124,Z 381.712,A -85,B 0,C 180,E1 -3268.098,E2 -3268.098} C_VEL
LIN {X 0,Y 552.109,Z 381.714,A -85,B 0,C 180,E1 -3270.609,E2 -3270.609} C_VEL
LIN {X 0,Y 552.12,Z 381.714,A -85,B 0,C 180,E1 -3273.186,E2 -3273.186} C_VEL
LIN {X 0,Y 552.107,Z 381.715,A -85,B 0,C 180,E1 -3275.842,E2 -3275.842} C_VEL
LIN {X 0,Y 552.124,Z 381.714,A -85,B 0,C 180,E1 -3279.062,E2 -3279.062} C_VEL
LIN {X 0,Y 552.138,Z 381.712,A -85,B 0,C 180,E1 -3281.445,E2 -3281.445} C_VEL
LIN {X 0,Y 552.093,Z 381.718,A -85,B 0,C 180,E1 -3284.532,E2 -3284.532} C_VEL
LIN {X 0,Y 552.13,Z 381.713,A -85,B 0,C 180,E1 -3287.585,E2 -3287.585} C_VEL
LIN {X 0,Y 552.133,Z 381.713,A -85,B 0,C 180,E1 -3290.474,E2 -3290.474} C_VEL
LIN {X 0,Y 552.162,Z 381.711,A -85,B 0,C 180,E1 -3292.916,E2 -3292.916} C_VEL
LIN {X 0,Y 552.65,Z 385.504,A -85,B 0,C 180,E1 -3294.477,E2 -3294.477} C_VEL
LIN {X 0,Y 552.575,Z 392.321,A -85,B 0,C 180,E1 -3297.08,E2 -3297.08} C_VEL
LIN {X 0,Y 552.373,Z 400.079,A -85,B 0,C 180,E1 -3299.904,E2 -3299.904} C_VEL
LIN {X 0,Y 552.238,Z 409.021,A -85,B 0,C 180,E1 -3302.98,E2 -3302.98} C_VEL
LIN {X 0,Y 552.157,Z 416.696,A -85,B 0,C 180,E1 -3305.565,E2 -3305.565} C_VEL
LIN {X 0,Y 552.082,Z 425.091,A -85,B 0,C 180,E1 -3308.336,E2 -3308.336} C_VEL
LIN {X 0,Y 552.026,Z 433.628,A -85,B 0,C 180,E1 -3311.056,E2 -3311.056} C_VEL
LIN {X 0,Y 551.929,Z 441.911,A -85,B 0,C 180,E1 -3313.732,E2 -3313.732} C_VEL
LIN {X 0,Y 551.896,Z 450.195,A -85,B 0,C 180,E1 -3316.374,E2 -3316.374} C_VEL
LIN {X 0,Y 551.873,Z 452.192,A -85,B 0,C 180,E1 -3317.006,E2 -3317.006} C_VEL
LIN {X 0,Y 553.073,Z 460.536,A -85,B 0,C 180,E1 -3317.198,E2 -3317.198} C_VEL
LIN {X 0,Y 552.946,Z 473.185,A -85,B 0,C 180,E1 -3317.569,E2 -3317.569} C_VEL
LIN {X 0,Y 552.743,Z 485.499,A -85,B 0,C 180,E1 -3318.076,E2 -3318.076} C_VEL
LIN {X 0,Y 552.579,Z 497.181,A -85,B 0,C 180,E1 -3318.714,E2 -3318.714} C_VEL
LIN {X 0,Y 552.433,Z 507.926,A -85,B 0,C 180,E1 -3319.463,E2 -3319.463} C_VEL
LIN {X 0,Y 552.233,Z 517.603,A -85,B 0,C 180,E1 -3320.292,E2 -3320.292} C_VEL
LIN {X 0,Y 552.079,Z 526.416,A -85,B 0,C 180,E1 -3321.213,E2 -3321.213} C_VEL
LIN {X 0,Y 551.949,Z 535.005,A -85,B 0,C 180,E1 -3322.317,E2 -3322.317} C_VEL
LIN {X 0,Y 551.823,Z 541.87,A -85,B 0,C 180,E1 -3323.418,E2 -3323.418} C_VEL
LIN {X 0,Y 551.804,Z 547.367,A -85,B 0,C 180,E1 -3324.519,E2 -3324.519} C_VEL
LIN {X 0,Y 551.764,Z 551.678,A -85,B 0,C 180,E1 -3325.617,E2 -3325.617} C_VEL
LIN {X 0,Y 551.75,Z 553.959,A -85,B 0,C 180,E1 -3326.349,E2 -3326.349} C_VEL
LIN {X 0,Y 551.723,Z 555.808,A -85,B 0,C 180,E1 -3327.08,E2 -3327.08} C_VEL
LIN {X 0,Y 551.645,Z 558.185,A -85,B 0,C 180,E1 -3328.54,E2 -3328.54} C_VEL
LIN {X 0,Y 551.64,Z 559,A -85,B 0,C 180,E1 -3330,E2 -3330} C_VEL
LIN {X 0,Y 551.645,Z 558.185,A -85,B 0,C 180,E1 -3331.46,E2 -3331.46} C_VEL
LIN {X 0,Y 551.723,Z 555.809,A -85,B 0,C 180,E1 -3332.921,E2 -3332.921} C_VEL
LIN {X 0,Y 551.764,Z 552.895,A -85,B 0,C 180,E1 -3334.017,E2 -3334.017} C_VEL
LIN {X 0,Y 551.724,Z 548.948,A -85,B 0,C 180,E1 -3335.116,E2 -3335.116} C_VEL
LIN {X 0,Y 551.803,Z 543.189,A -85,B 0,C 180,E1 -3336.341,E2 -3336.341} C_VEL
LIN {X 0,Y 551.927,Z 536.235,A -85,B 0,C 180,E1 -3337.5,E2 -3337.5} C_VEL
LIN {X 0,Y 552.082,Z 527.989,A -85,B 0,C 180,E1 -3338.603,E2 -3338.603} C_VEL
LIN {X 0,Y 552.201,Z 519.537,A -85,B 0,C 180,E1 -3339.524,E2 -3339.524} C_VEL
LIN {X 0,Y 552.397,Z 509.092,A -85,B 0,C 180,E1 -3340.446,E2 -3340.446} C_VEL
LIN {X 0,Y 552.594,Z 497.276,A -85,B 0,C 180,E1 -3341.28,E2 -3341.28} C_VEL
LIN {X 0,Y 552.742,Z 485.485,A -85,B 0,C 180,E1 -3341.924,E2 -3341.924} C_VEL
LIN {X 0,Y 552.946,Z 473.162,A -85,B 0,C 180,E1 -3342.432,E2 -3342.432} C_VEL
LIN {X 0,Y 553.073,Z 460.509,A -85,B 0,C 180,E1 -3342.802,E2 -3342.802} C_VEL
LIN {X 0,Y 551.872,Z 452.19,A -85,B 0,C 180,E1 -3342.994,E2 -3342.994} C_VEL
LIN {X 0,Y 551.915,Z 443.093,A -85,B 0,C 180,E1 -3345.889,E2 -3345.889} C_VEL
LIN {X 0,Y 552,Z 434.81,A -85,B 0,C 180,E1 -3348.56,E2 -3348.56} C_VEL
LIN {X 0,Y 552.083,Z 426.377,A -85,B 0,C 180,E1 -3351.273,E2 -3351.273} C_VEL
LIN {X 0,Y 552.172,Z 418.015,A -85,B 0,C 180,E1 -3354.035,E2 -3354.035} C_VEL
LIN {X 0,Y 552.275,Z 409.182,A -85,B 0,C 180,E1 -3357.027,E2 -3357.027} C_VEL
LIN {X 0,Y 552.396,Z 400.263,A -85,B 0,C 180,E1 -3360.1,E2 -3360.1} C_VEL
LIN {X 0,Y 552.59,Z 391.863,A -85,B 0,C 180,E1 -3363.154,E2 -3363.154} C_VEL
LIN {X 0,Y 552.654,Z 385.616,A -85,B 0,C 180,E1 -3365.523,E2 -3365.523} C_VEL
LIN {X 0,Y 552.164,Z 381.709,A -85,B 0,C 180,E1 -3367.085,E2 -3367.085} C_VEL
LIN {X 0,Y 552.117,Z 381.714,A -85,B 0,C 180,E1 -3370.204,E2 -3370.204} C_VEL
LIN {X 0,Y 552.133,Z 381.713,A -85,B 0,C 180,E1 -3372.425,E2 -3372.425} C_VEL
LIN {X 0,Y 552.097,Z 381.715,A -85,B 0,C 180,E1 -3375.562,E2 -3375.562} C_VEL
LIN {X 0,Y 552.122,Z 381.713,A -85,B 0,C 180,E1 -3378.554,E2 -3378.554} C_VEL
LIN {X 0,Y 552.119,Z 381.712,A -85,B 0,C 180,E1 -3381.411,E2 -3381.411} C_VEL
LIN {X 0,Y 552.103,Z 381.716,A -85,B 0,C 180,E1 -3384.157,E2 -3384.157} C_VEL
LIN {X 0,Y 552.108,Z 381.715,A -85,B 0,C 180,E1 -3386.813,E2 -3386.813} C_VEL
LIN {X 0,Y 552.104,Z 381.714,A -85,B 0,C 180,E1 -3389.391,E2 -3389.391} C_VEL
LIN {X 0,Y 552.11,Z 381.712,A -85,B 0,C 180,E1 -3391.902,E2 -3391.902} C_VEL
LIN {X 0,Y 552.156,Z 381.707,A -85,B 0,C 180,E1 -3394.65,E2 -3394.65} C_VEL
LIN {X 0,Y 552.094,Z 381.716,A -85,B 0,C 180,E1 -3397.549,E2 -3397.549} C_VEL
LIN {X 0,Y 552.145,Z 381.708,A -85,B 0,C 180,E1 -3400.375,E2 -3400.375} C_VEL
LIN {X 0,Y 552.156,Z 381.708,A -85,B 0,C 180,E1 -3402.977,E2 -3402.977} C_VEL
LIN {X 0,Y 552.135,Z 381.71,A -85,B 0,C 180,E1 -3406.004,E2 -3406.004} C_VEL
LIN {X 0,Y 552.162,Z 381.707,A -85,B 0,C 180,E1 -3408.993,E2 -3408.993} C_VEL
LIN {X 0,Y 552.159,Z 381.707,A -85,B 0,C 180,E1 -3411.951,E2 -3411.951} C_VEL
LIN {X 0,Y 552.229,Z 381.699,A -85,B 0,C 180,E1 -3414.889,E2 -3414.889} C_VEL
LIN {X 0,Y 552.219,Z 381.701,A -85,B 0,C 180,E1 -3417.812,E2 -3417.812} C_VEL
LIN {X 0,Y 552.242,Z 381.697,A -85,B 0,C 180,E1 -3420.729,E2 -3420.729} C_VEL
LIN {X 0,Y 552.209,Z 381.701,A -85,B 0,C 180,E1 -3422.918,E2 -3422.918} C_VEL
LIN {X 0,Y 552.199,Z 381.704,A -85,B 0,C 180,E1 -3425.844,E2 -3425.844} C_VEL
LIN {X 0,Y 552.162,Z 381.707,A -85,B 0,C 180,E1 -3428.786,E2 -3428.786} C_VEL
LIN {X 0,Y 552.163,Z 381.708,A -85,B 0,C 180,E1 -3431.75,E2 -3431.75} C_VEL
LIN {X 0,Y 552.137,Z 381.71,A -85,B 0,C 180,E1 -3434.748,E2 -3434.748} C_VEL
LIN {X 0,Y 552.113,Z 381.714,A -85,B 0,C 180,E1 -3437.788,E2 -3437.788} C_VEL
LIN {X 0,Y 552.127,Z 381.711,A -85,B 0,C 180,E1 -3440.101,E2 -3440.101} C_VEL
LIN {X 0,Y 552.092,Z 381.716,A -85,B 0,C 180,E1 -3442.451,E2 -3442.451} C_VEL
LIN {X 0,Y 552.155,Z 381.707,A -85,B 0,C 180,E1 -3445.35,E2 -3445.35} C_VEL
LIN {X 0,Y 552.12,Z 381.711,A -85,B 0,C 180,E1 -3448.098,E2 -3448.098} C_VEL
LIN {X 0,Y 552.103,Z 381.714,A -85,B 0,C 180,E1 -3450.609,E2 -3450.609} C_VEL
LIN {X 0,Y 552.124,Z 381.712,A -85,B 0,C 180,E1 -3453.185,E2 -3453.185} C_VEL
LIN {X 0,Y 552.114,Z 381.711,A -85,B 0,C 180,E1 -3453.788,E2 -3453.788} C_VEL
LIN {X 0,Y 551.477,Z 381.793,A -85,B 0,C 180,E1 -3454.397,E2 -3454.397} C_VEL
LIN {X 0,Y 548.657,Z 382.148,A -85,B 0,C 180,E1 -3455.385,E2 -3455.385} C_VEL
LIN {X 0,Y 546.238,Z 382.451,A -85,B 0,C 180,E1 -3456.181,E2 -3456.181} C_VEL
LIN {X 0,Y 545.169,Z 382.581,A -85,B 0,C 180,E1 -3456.795,E2 -3456.795} C_VEL
LIN {X 0,Y 545.067,Z 382.592,A -85,B 0,C 180,E1 -3457.003,E2 -3457.003} C_VEL
LIN {X 0,Y 545.066,Z 382.59,A -85,B 0,C 180,E1 -3460.143,E2 -3460.143} C_VEL
LIN {X 0,Y 545.079,Z 382.59,A -85,B 0,C 180,E1 -3463.107,E2 -3463.107} C_VEL
LIN {X 0,Y 545.05,Z 382.593,A -85,B 0,C 180,E1 -3466.226,E2 -3466.226} C_VEL
LIN {X 0,Y 545.095,Z 382.59,A -85,B 0,C 180,E1 -3468.887,E2 -3468.887} C_VEL
LIN {X 0,Y 545.051,Z 382.592,A -85,B 0,C 180,E1 -3471.763,E2 -3471.763} C_VEL
LIN {X 0,Y 545.055,Z 382.592,A -85,B 0,C 180,E1 -3474.533,E2 -3474.533} C_VEL
LIN {X 0,Y 545.071,Z 382.592,A -85,B 0,C 180,E1 -3477.212,E2 -3477.212} C_VEL
LIN {X 0,Y 545.065,Z 382.593,A -85,B 0,C 180,E1 -3479.81,E2 -3479.81} C_VEL
LIN {X 0,Y 545.079,Z 382.59,A -85,B 0,C 180,E1 -3482.344,E2 -3482.344} C_VEL
LIN {X 0,Y 545.12,Z 382.584,A -85,B 0,C 180,E1 -3484.82,E2 -3484.82} C_VEL
LIN {X 0,Y 545.04,Z 382.593,A -85,B 0,C 180,E1 -3487.242,E2 -3487.242} C_VEL
LIN {X 0,Y 545.12,Z 382.587,A -85,B 0,C 180,E1 -3490.415,E2 -3490.415} C_VEL
LIN {X 0,Y 545.065,Z 382.589,A -85,B 0,C 180,E1 -3493.521,E2 -3493.521} C_VEL
LIN {X 0,Y 545.097,Z 382.586,A -85,B 0,C 180,E1 -3495.82,E2 -3495.82} C_VEL
LIN {X 0,Y 545.12,Z 382.585,A -85,B 0,C 180,E1 -3498.849,E2 -3498.849} C_VEL
LIN {X 0,Y 545.128,Z 382.582,A -85,B 0,C 180,E1 -3501.847,E2 -3501.847} C_VEL
LIN {X 0,Y 545.204,Z 382.575,A -85,B 0,C 180,E1 -3504.823,E2 -3504.823} C_VEL
LIN {X 0,Y 545.2,Z 382.573,A -85,B 0,C 180,E1 -3507.783,E2 -3507.783} C_VEL
LIN {X 0,Y 545.215,Z 382.574,A -85,B 0,C 180,E1 -3510.738,E2 -3510.738} C_VEL
LIN {X 0,Y 545.172,Z 382.579,A -85,B 0,C 180,E1 -3512.955,E2 -3512.955} C_VEL
LIN {X 0,Y 545.168,Z 382.578,A -85,B 0,C 180,E1 -3515.919,E2 -3515.919} C_VEL
LIN {X 0,Y 545.002,Z 382.602,A -85,B 0,C 180,E1 -3518.155,E2 -3518.155} C_VEL
LIN {X 0,Y 544.957,Z 383.253,A -85,B 0,C 180,E1 -3518.902,E2 -3518.902} C_VEL
LIN {X 0,Y 544.895,Z 387.588,A -85,B 0,C 180,E1 -3521.909,E2 -3521.909} C_VEL
LIN {X 0,Y 544.808,Z 392.047,A -85,B 0,C 180,E1 -3524.951,E2 -3524.951} C_VEL
LIN {X 0,Y 544.737,Z 396.606,A -85,B 0,C 180,E1 -3528.037,E2 -3528.037} C_VEL
LIN {X 0,Y 544.656,Z 400.125,A -85,B 0,C 180,E1 -3530.389,E2 -3530.389} C_VEL
LIN {X 0,Y 544.634,Z 403.694,A -85,B 0,C 180,E1 -3532.775,E2 -3532.775} C_VEL
LIN {X 0,Y 544.636,Z 407.714,A -85,B 0,C 180,E1 -3535.407,E2 -3535.407} C_VEL
LIN {X 0,Y 544.569,Z 411.287,A -85,B 0,C 180,E1 -3537.684,E2 -3537.684} C_VEL
LIN {X 0,Y 544.591,Z 414.909,A -85,B 0,C 180,E1 -3539.909,E2 -3539.909} C_VEL
LIN {X 0,Y 546.104,Z 424.947,A -85,B 0,C 180,E1 -3540.191,E2 -3540.191} C_VEL
LIN {X 0,Y 545.959,Z 436.596,A -85,B 0,C 180,E1 -3540.578,E2 -3540.578} C_VEL
LIN {X 0,Y 545.692,Z 448.464,A -85,B 0,C 180,E1 -3541.115,E2 -3541.115} C_VEL
LIN {X 0,Y 545.469,Z 460.362,A -85,B 0,C 180,E1 -3541.82,E2 -3541.82} C_VEL
LIN {X 0,Y 545.291,Z 471.551,A -85,B 0,C 180,E1 -3542.663,E2 -3542.663} C_VEL
LIN {X 0,Y 545.111,Z 482.137,A -85,B 0,C 180,E1 -3543.668,E2 -3543.668} C_VEL
LIN {X 0,Y 544.953,Z 489.92,A -85,B 0,C 180,E1 -3544.572,E2 -3544.572} C_VEL
LIN {X 0,Y 544.81,Z 497.511,A -85,B 0,C 180,E1 -3545.64,E2 -3545.64} C_VEL
LIN {X 0,Y 544.77,Z 503.266,A -85,B 0,C 180,E1 -3546.636,E2 -3546.636} C_VEL
LIN {X 0,Y 544.683,Z 508.294,A -85,B 0,C 180,E1 -3547.706,E2 -3547.706} C_VEL
LIN {X 0,Y 544.648,Z 512.139,A -85,B 0,C 180,E1 -3548.743,E2 -3548.743} C_VEL
LIN {X 0,Y 544.603,Z 516.007,A -85,B 0,C 180,E1 -3550.183,E2 -3550.183} C_VEL
LIN {X 0,Y 544.573,Z 518.154,A -85,B 0,C 180,E1 -3551.538,E2 -3551.538} C_VEL
LIN {X 0,Y 544.544,Z 518.919,A -85,B 0,C 180,E1 -3552.637,E2 -3552.637} C_VEL
LIN {X 0,Y 544.58,Z 518.531,A -85,B 0,C 180,E1 -3554.177,E2 -3554.177} C_VEL
LIN {X 0,Y 544.586,Z 517.266,A -85,B 0,C 180,E1 -3555.217,E2 -3555.217} C_VEL
LIN {X 0,Y 544.602,Z 515.163,A -85,B 0,C 180,E1 -3556.275,E2 -3556.275} C_VEL
LIN {X 0,Y 544.653,Z 512.133,A -85,B 0,C 180,E1 -3557.349,E2 -3557.349} C_VEL
LIN {X 0,Y 544.707,Z 508.028,A -85,B 0,C 180,E1 -3558.446,E2 -3558.446} C_VEL
LIN {X 0,Y 544.722,Z 502.639,A -85,B 0,C 180,E1 -3559.571,E2 -3559.571} C_VEL
LIN {X 0,Y 544.863,Z 495.197,A -85,B 0,C 180,E1 -3560.8,E2 -3560.8} C_VEL
LIN {X 0,Y 545.035,Z 487.121,A -85,B 0,C 180,E1 -3561.865,E2 -3561.865} C_VEL
LIN {X 0,Y 545.214,Z 477.285,A -85,B 0,C 180,E1 -3562.909,E2 -3562.909} C_VEL
LIN {X 0,Y 545.387,Z 466.774,A -85,B 0,C 180,E1 -3563.812,E2 -3563.812} C_VEL
LIN {X 0,Y 545.614,Z 455.567,A -85,B 0,C 180,E1 -3564.575,E2 -3564.575} C_VEL
LIN {X 0,Y 545.795,Z 442.788,A -85,B 0,C 180,E1 -3565.251,E2 -3565.251} C_VEL
LIN {X 0,Y 546.052,Z 430.097,A -85,B 0,C 180,E1 -3565.743,E2 -3565.743} C_VEL
LIN {X 0,Y 545.918,Z 422.646,A -85,B 0,C 180,E1 -3565.963,E2 -3565.963} C_VEL
LIN {X 0,Y 544.624,Z 414.891,A -85,B 0,C 180,E1 -3566.191,E2 -3566.191} C_VEL
LIN {X 0,Y 544.604,Z 410.457,A -85,B 0,C 180,E1 -3568.923,E2 -3568.923} C_VEL
LIN {X 0,Y 544.654,Z 406.542,A -85,B 0,C 180,E1 -3571.482,E2 -3571.482} C_VEL
LIN {X 0,Y 544.701,Z 402.806,A -85,B 0,C 180,E1 -3573.98,E2 -3573.98} C_VEL
LIN {X 0,Y 544.77,Z 399.233,A -85,B 0,C 180,E1 -3576.426,E2 -3576.426} C_VEL
LIN {X 0,Y 544.838,Z 395.775,A -85,B 0,C 180,E1 -3578.827,E2 -3578.827} C_VEL
LIN {X 0,Y 544.835,Z 392.204,A -85,B 0,C 180,E1 -3581.187,E2 -3581.187} C_VEL
LIN {X 0,Y 544.882,Z 388.832,A -85,B 0,C 180,E1 -3583.515,E2 -3583.515} C_VEL
LIN {X 0,Y 544.965,Z 385.567,A -85,B 0,C 180,E1 -3585.816,E2 -3585.816} C_VEL
LIN {X 0,Y 544.965,Z 383.381,A -85,B 0,C 180,E1 -3587.336,E2 -3587.336} C_VEL
LIN {X 0,Y 544.996,Z 382.603,A -85,B 0,C 180,E1 -3588.093,E2 -3588.093} C_VEL
LIN {X 0,Y 545.099,Z 382.591,A -85,B 0,C 180,E1 -3590.351,E2 -3590.351} C_VEL
LIN {X 0,Y 545.156,Z 382.58,A -85,B 0,C 180,E1 -3593.049,E2 -3593.049} C_VEL
LIN {X 0,Y 545.204,Z 382.574,A -85,B 0,C 180,E1 -3594.823,E2 -3594.823} C_VEL
LIN {X 0,Y 545.19,Z 382.577,A -85,B 0,C 180,E1 -3597.784,E2 -3597.784} C_VEL
LIN {X 0,Y 545.213,Z 382.575,A -85,B 0,C 180,E1 -3600.739,E2 -3600.739} C_VEL
LIN {X 0,Y 545.169,Z 382.58,A -85,B 0,C 180,E1 -3602.956,E2 -3602.956} C_VEL
LIN {X 0,Y 545.17,Z 382.58,A -85,B 0,C 180,E1 -3605.92,E2 -3605.92} C_VEL
LIN {X 0,Y 545.118,Z 382.586,A -85,B 0,C 180,E1 -3608.9,E2 -3608.9} C_VEL
LIN {X 0,Y 545.131,Z 382.584,A -85,B 0,C 180,E1 -3611.904,E2 -3611.904} C_VEL
LIN {X 0,Y 545.082,Z 382.589,A -85,B 0,C 180,E1 -3614.944,E2 -3614.944} C_VEL
LIN {X 0,Y 545.08,Z 382.589,A -85,B 0,C 180,E1 -3618.026,E2 -3618.026} C_VEL
LIN {X 0,Y 545.096,Z 382.589,A -85,B 0,C 180,E1 -3620.372,E2 -3620.372} C_VEL
LIN {X 0,Y 545.088,Z 382.591,A -85,B 0,C 180,E1 -3623.559,E2 -3623.559} C_VEL
LIN {X 0,Y 545.085,Z 382.589,A -85,B 0,C 180,E1 -3626,E2 -3626} C_VEL
LIN {X 0,Y 545.09,Z 382.59,A -85,B 0,C 180,E1 -3628.749,E2 -3628.749} C_VEL
LIN {X 0,Y 545.067,Z 382.592,A -85,B 0,C 180,E1 -3631.048,E2 -3631.048} C_VEL
LIN {X 0,Y 545.067,Z 382.591,A -85,B 0,C 180,E1 -3633.672,E2 -3633.672} C_VEL
LIN {X 0,Y 545.052,Z 382.594,A -85,B 0,C 180,E1 -3636.38,E2 -3636.38} C_VEL
LIN {X 0,Y 545.104,Z 382.589,A -85,B 0,C 180,E1 -3639.325,E2 -3639.325} C_VEL
LIN {X 0,Y 545.081,Z 382.591,A -85,B 0,C 180,E1 -3642.103,E2 -3642.103} C_VEL
LIN {X 0,Y 545.059,Z 382.593,A -85,B 0,C 180,E1 -3645.168,E2 -3645.168} C_VEL
LIN {X 0,Y 545.082,Z 382.589,A -85,B 0,C 180,E1 -3647.898,E2 -3647.898} C_VEL
LIN {X 0,Y 545.105,Z 382.589,A -85,B 0,C 180,E1 -3650.676,E2 -3650.676} C_VEL
LIN {X 0,Y 545.137,Z 382.691,A -85,B 0,C 180,E1 -3652.756,E2 -3652.756} C_VEL
LIN {X 0,Y 545.659,Z 387.074,A -85,B 0,C 180,E1 -3654.579,E2 -3654.579} C_VEL
LIN {X 0,Y 545.579,Z 392.932,A -85,B 0,C 180,E1 -3656.858,E2 -3656.858} C_VEL
LIN {X 0,Y 545.358,Z 400.914,A -85,B 0,C 180,E1 -3659.829,E2 -3659.829} C_VEL
LIN {X 0,Y 545.228,Z 409.392,A -85,B 0,C 180,E1 -3662.8,E2 -3662.8} C_VEL
LIN {X 0,Y 545.104,Z 417.701,A -85,B 0,C 180,E1 -3665.634,E2 -3665.634} C_VEL
LIN {X 0,Y 545.032,Z 425.317,A -85,B 0,C 180,E1 -3668.19,E2 -3668.19} C_VEL
LIN {X 0,Y 544.937,Z 434.652,A -85,B 0,C 180,E1 -3671.191,E2 -3671.191} C_VEL
LIN {X 0,Y 544.851,Z 443.095,A -85,B 0,C 180,E1 -3673.9,E2 -3673.9} C_VEL
LIN {X 0,Y 544.766,Z 452.192,A -85,B 0,C 180,E1 -3676.834,E2 -3676.834} C_VEL
LIN {X 0,Y 546.156,Z 461.451,A -85,B 0,C 180,E1 -3677.057,E2 -3677.057} C_VEL
LIN {X 0,Y 545.993,Z 474.485,A -85,B 0,C 180,E1 -3677.455,E2 -3677.455} C_VEL
LIN {X 0,Y 545.787,Z 485.499,A -85,B 0,C 180,E1 -3677.922,E2 -3677.922} C_VEL
LIN {X 0,Y 545.595,Z 497.592,A -85,B 0,C 180,E1 -3678.595,E2 -3678.595} C_VEL
LIN {X 0,Y 545.42,Z 509.098,A -85,B 0,C 180,E1 -3679.42,E2 -3679.42} C_VEL
LIN {X 0,Y 545.165,Z 519.543,A -85,B 0,C 180,E1 -3680.353,E2 -3680.353} C_VEL
LIN {X 0,Y 545.029,Z 527.994,A -85,B 0,C 180,E1 -3681.286,E2 -3681.286} C_VEL
LIN {X 0,Y 544.859,Z 536.238,A -85,B 0,C 180,E1 -3682.403,E2 -3682.403} C_VEL
LIN {X 0,Y 544.734,Z 543.614,A -85,B 0,C 180,E1 -3683.655,E2 -3683.655} C_VEL
LIN {X 0,Y 544.653,Z 548.951,A -85,B 0,C 180,E1 -3684.818,E2 -3684.818} C_VEL
LIN {X 0,Y 544.684,Z 552.896,A -85,B 0,C 180,E1 -3685.931,E2 -3685.931} C_VEL
LIN {X 0,Y 544.65,Z 555.808,A -85,B 0,C 180,E1 -3687.042,E2 -3687.042} C_VEL
LIN {X 0,Y 544.546,Z 558.184,A -85,B 0,C 180,E1 -3688.521,E2 -3688.521} C_VEL
LIN {X 0,Y 544.541,Z 559,A -85,B 0,C 180,E1 -3690,E2 -3690} C_VEL
LIN {X 0,Y 544.546,Z 558.184,A -85,B 0,C 180,E1 -3691.479,E2 -3691.479} C_VEL
LIN {X 0,Y 544.65,Z 555.809,A -85,B 0,C 180,E1 -3692.959,E2 -3692.959} C_VEL
LIN {X 0,Y 544.684,Z 552.895,A -85,B 0,C 180,E1 -3694.07,E2 -3694.07} C_VEL
LIN {X 0,Y 544.653,Z 548.947,A -85,B 0,C 180,E1 -3695.183,E2 -3695.183} C_VEL
LIN {X 0,Y 544.74,Z 543.704,A -85,B 0,C 180,E1 -3696.328,E2 -3696.328} C_VEL
LIN {X 0,Y 544.837,Z 537.466,A -85,B 0,C 180,E1 -3697.412,E2 -3697.412} C_VEL
LIN {X 0,Y 545.007,Z 529.476,A -85,B 0,C 180,E1 -3698.528,E2 -3698.528} C_VEL
LIN {X 0,Y 545.142,Z 521.332,A -85,B 0,C 180,E1 -3699.461,E2 -3699.461} C_VEL
LIN {X 0,Y 545.35,Z 511.396,A -85,B 0,C 180,E1 -3700.394,E2 -3700.394} C_VEL
LIN {X 0,Y 545.542,Z 501.587,A -85,B 0,C 180,E1 -3701.142,E2 -3701.142} C_VEL
LIN {X 0,Y 545.687,Z 490.657,A -85,B 0,C 180,E1 -3701.813,E2 -3701.813} C_VEL
LIN {X 0,Y 545.899,Z 478.099,A -85,B 0,C 180,E1 -3702.406,E2 -3702.406} C_VEL
LIN {X 0,Y 546.127,Z 465.08,A -85,B 0,C 180,E1 -3702.85,E2 -3702.85} C_VEL
LIN {X 0,Y 545.896,Z 459.065,A -85,B 0,C 180,E1 -3703.006,E2 -3703.006} C_VEL
LIN {X 0,Y 544.784,Z 452.116,A -85,B 0,C 180,E1 -3703.19,E2 -3703.19} C_VEL
LIN {X 0,Y 544.851,Z 443.093,A -85,B 0,C 180,E1 -3706.101,E2 -3706.101} C_VEL
LIN {X 0,Y 544.94,Z 434.694,A -85,B 0,C 180,E1 -3708.81,E2 -3708.81} C_VEL
LIN {X 0,Y 545.071,Z 425.394,A -85,B 0,C 180,E1 -3711.821,E2 -3711.821} C_VEL
LIN {X 0,Y 545.153,Z 416.695,A -85,B 0,C 180,E1 -3714.77,E2 -3714.77} C_VEL
LIN {X 0,Y 545.277,Z 408.404,A -85,B 0,C 180,E1 -3717.646,E2 -3717.646} C_VEL
LIN {X 0,Y 545.426,Z 399.908,A -85,B 0,C 180,E1 -3720.623,E2 -3720.623} C_VEL
LIN {X 0,Y 545.626,Z 391.822,A -85,B 0,C 180,E1 -3723.633,E2 -3723.633} C_VEL
LIN {X 0,Y 545.664,Z 386.301,A -85,B 0,C 180,E1 -3725.765,E2 -3725.765} C_VEL
LIN {X 0,Y 545.107,Z 382.587,A -85,B 0,C 180,E1 -3727.298,E2 -3727.298} C_VEL
LIN {X 0,Y 545.07,Z 382.592,A -85,B 0,C 180,E1 -3730.142,E2 -3730.142} C_VEL
LIN {X 0,Y 545.08,Z 382.589,A -85,B 0,C 180,E1 -3733.106,E2 -3733.106} C_VEL
LIN {X 0,Y 545.051,Z 382.592,A -85,B 0,C 180,E1 -3736.226,E2 -3736.226} C_VEL
LIN {X 0,Y 545.082,Z 382.588,A -85,B 0,C 180,E1 -3738.885,E2 -3738.885} C_VEL
LIN {X 0,Y 545.054,Z 382.594,A -85,B 0,C 180,E1 -3741.763,E2 -3741.763} C_VEL
LIN {X 0,Y 545.053,Z 382.593,A -85,B 0,C 180,E1 -3744.533,E2 -3744.533} C_VEL
LIN {X 0,Y 545.066,Z 382.59,A -85,B 0,C 180,E1 -3747.211,E2 -3747.211} C_VEL
LIN {X 0,Y 545.065,Z 382.591,A -85,B 0,C 180,E1 -3749.81,E2 -3749.81} C_VEL
LIN {X 0,Y 545.082,Z 382.589,A -85,B 0,C 180,E1 -3752.344,E2 -3752.344} C_VEL
LIN {X 0,Y 545.118,Z 382.585,A -85,B 0,C 180,E1 -3754.82,E2 -3754.82} C_VEL
LIN {X 0,Y 545.039,Z 382.596,A -85,B 0,C 180,E1 -3757.242,E2 -3757.242} C_VEL
LIN {X 0,Y 545.117,Z 382.583,A -85,B 0,C 180,E1 -3760.415,E2 -3760.415} C_VEL
LIN {X 0,Y 545.073,Z 382.59,A -85,B 0,C 180,E1 -3763.521,E2 -3763.521} C_VEL
LIN {X 0,Y 545.095,Z 382.588,A -85,B 0,C 180,E1 -3765.82,E2 -3765.82} C_VEL
LIN {X 0,Y 545.118,Z 382.584,A -85,B 0,C 180,E1 -3768.849,E2 -3768.849} C_VEL
LIN {X 0,Y 545.13,Z 382.584,A -85,B 0,C 180,E1 -3771.847,E2 -3771.847} C_VEL
LIN {X 0,Y 545.204,Z 382.573,A -85,B 0,C 180,E1 -3774.823,E2 -3774.823} C_VEL
LIN {X 0,Y 545.191,Z 382.576,A -85,B 0,C 180,E1 -3777.784,E2 -3777.784} C_VEL
LIN {X 0,Y 545.212,Z 382.572,A -85,B 0,C 180,E1 -3780.739,E2 -3780.739} C_VEL
LIN {X 0,Y 545.175,Z 382.577,A -85,B 0,C 180,E1 -3782.956,E2 -3782.956} C_VEL
LIN {X 0,Y 545.171,Z 382.579,A -85,B 0,C 180,E1 -3785.919,E2 -3785.919} C_VEL
LIN {X 0,Y 545.121,Z 382.584,A -85,B 0,C 180,E1 -3788.9,E2 -3788.9} C_VEL
LIN {X 0,Y 545.135,Z 382.583,A -85,B 0,C 180,E1 -3791.904,E2 -3791.904} C_VEL
LIN {X 0,Y 545.086,Z 382.588,A -85,B 0,C 180,E1 -3794.944,E2 -3794.944} C_VEL
LIN {X 0,Y 545.081,Z 382.591,A -85,B 0,C 180,E1 -3798.026,E2 -3798.026} C_VEL
LIN {X 0,Y 545.093,Z 382.59,A -85,B 0,C 180,E1 -3800.372,E2 -3800.372} C_VEL
LIN {X 0,Y 545.082,Z 382.589,A -85,B 0,C 180,E1 -3803.559,E2 -3803.559} C_VEL
LIN {X 0,Y 545.079,Z 382.589,A -85,B 0,C 180,E1 -3806.001,E2 -3806.001} C_VEL
LIN {X 0,Y 545.089,Z 382.59,A -85,B 0,C 180,E1 -3808.748,E2 -3808.748} C_VEL
LIN {X 0,Y 545.06,Z 382.59,A -85,B 0,C 180,E1 -3811.679,E2 -3811.679} C_VEL
LIN {X 0,Y 545.078,Z 382.591,A -85,B 0,C 180,E1 -3814.563,E2 -3814.563} C_VEL
LIN {X 0,Y 545.067,Z 382.592,A -85,B 0,C 180,E1 -3817.003,E2 -3817.003} C_VEL
LIN {X 0,Y 544.357,Z 382.678,A -85,B 0,C 180,E1 -3817.619,E2 -3817.619} C_VEL
LIN {X 0,Y 541.49,Z 383.036,A -85,B 0,C 180,E1 -3818.62,E2 -3818.62} C_VEL
LIN {X 0,Y 539.102,Z 383.335,A -85,B 0,C 180,E1 -3819.426,E2 -3819.426} C_VEL
LIN {X 0,Y 538.092,Z 383.459,A -85,B 0,C 180,E1 -3820.048,E2 -3820.048} C_VEL
LIN {X 0,Y 538.017,Z 383.467,A -85,B 0,C 180,E1 -3820.258,E2 -3820.258} C_VEL
LIN {X 0,Y 538.027,Z 383.47,A -85,B 0,C 180,E1 -3822.988,E2 -3822.988} C_VEL
LIN {X 0,Y 538.004,Z 383.47,A -85,B 0,C 180,E1 -3826.184,E2 -3826.184} C_VEL
LIN {X 0,Y 538.051,Z 383.464,A -85,B 0,C 180,E1 -3829.253,E2 -3829.253} C_VEL
LIN {X 0,Y 537.992,Z 383.471,A -85,B 0,C 180,E1 -3832.122,E2 -3832.122} C_VEL
LIN {X 0,Y 538.014,Z 383.471,A -85,B 0,C 180,E1 -3834.917,E2 -3834.917} C_VEL
LIN {X 0,Y 538.02,Z 383.468,A -85,B 0,C 180,E1 -3837.617,E2 -3837.617} C_VEL
LIN {X 0,Y 538.019,Z 383.468,A -85,B 0,C 180,E1 -3840.239,E2 -3840.239} C_VEL
LIN {X 0,Y 538.057,Z 383.464,A -85,B 0,C 180,E1 -3842.796,E2 -3842.796} C_VEL
LIN {X 0,Y 538.051,Z 383.464,A -85,B 0,C 180,E1 -3845.293,E2 -3845.293} C_VEL
LIN {X 0,Y 538.025,Z 383.468,A -85,B 0,C 180,E1 -3848.546,E2 -3848.546} C_VEL
LIN {X 0,Y 538.036,Z 383.466,A -85,B 0,C 180,E1 -3850.94,E2 -3850.94} C_VEL
LIN {X 0,Y 538.018,Z 383.467,A -85,B 0,C 180,E1 -3853.299,E2 -3853.299} C_VEL
LIN {X 0,Y 538.066,Z 383.462,A -85,B 0,C 180,E1 -3855.631,E2 -3855.631} C_VEL
LIN {X 0,Y 538.08,Z 383.463,A -85,B 0,C 180,E1 -3858.701,E2 -3858.701} C_VEL
LIN {X 0,Y 538.085,Z 383.46,A -85,B 0,C 180,E1 -3861.739,E2 -3861.739} C_VEL
LIN {X 0,Y 538.163,Z 383.452,A -85,B 0,C 180,E1 -3864.755,E2 -3864.755} C_VEL
LIN {X 0,Y 538.171,Z 383.449,A -85,B 0,C 180,E1 -3867.754,E2 -3867.754} C_VEL
LIN {X 0,Y 538.185,Z 383.449,A -85,B 0,C 180,E1 -3870.748,E2 -3870.748} C_VEL
LIN {X 0,Y 538.139,Z 383.455,A -85,B 0,C 180,E1 -3872.994,E2 -3872.994} C_VEL
LIN {X 0,Y 538.119,Z 383.456,A -85,B 0,C 180,E1 -3875.997,E2 -3875.997} C_VEL
LIN {X 0,Y 537.943,Z 383.481,A -85,B 0,C 180,E1 -3878.262,E2 -3878.262} C_VEL
LIN {X 0,Y 537.85,Z 385.28,A -85,B 0,C 180,E1 -3879.78,E2 -3879.78} C_VEL
LIN {X 0,Y 537.814,Z 388.55,A -85,B 0,C 180,E1 -3882.068,E2 -3882.068} C_VEL
LIN {X 0,Y 537.746,Z 393.029,A -85,B 0,C 180,E1 -3885.152,E2 -3885.152} C_VEL
LIN {X 0,Y 537.693,Z 396.483,A -85,B 0,C 180,E1 -3887.495,E2 -3887.495} C_VEL
LIN {X 0,Y 537.649,Z 399.972,A -85,B 0,C 180,E1 -3889.868,E2 -3889.868} C_VEL
LIN {X 0,Y 537.559,Z 403.522,A -85,B 0,C 180,E1 -3892.28,E2 -3892.28} C_VEL
LIN {X 0,Y 537.533,Z 407.203,A -85,B 0,C 180,E1 -3894.732,E2 -3894.732} C_VEL
LIN {X 0,Y 537.51,Z 411.041,A -85,B 0,C 180,E1 -3897.238,E2 -3897.238} C_VEL
LIN {X 0,Y 537.487,Z 414.938,A -85,B 0,C 180,E1 -3899.739,E2 -3899.739} C_VEL
LIN {X 0,Y 539.176,Z 425.592,A -85,B 0,C 180,E1 -3900.041,E2 -3900.041} C_VEL
LIN {X 0,Y 538.995,Z 437.495,A -85,B 0,C 180,E1 -3900.452,E2 -3900.452} C_VEL
LIN {X 0,Y 538.702,Z 449.88,A -85,B 0,C 180,E1 -3901.035,E2 -3901.035} C_VEL
LIN {X 0,Y 538.489,Z 461.115,A -85,B 0,C 180,E1 -3901.723,E2 -3901.723} C_VEL
LIN {X 0,Y 538.3,Z 470.943,A -85,B 0,C 180,E1 -3902.474,E2 -3902.474} C_VEL
LIN {X 0,Y 538.137,Z 479.805,A -85,B 0,C 180,E1 -3903.297,E2 -3903.297} C_VEL
LIN {X 0,Y 537.947,Z 489.344,A -85,B 0,C 180,E1 -3904.387,E2 -3904.387} C_VEL
LIN {X 0,Y 537.767,Z 497.139,A -85,B 0,C 180,E1 -3905.485,E2 -3905.485} C_VEL
LIN {X 0,Y 537.67,Z 504.162,A -85,B 0,C 180,E1 -3906.727,E2 -3906.727} C_VEL
LIN {X 0,Y 537.572,Z 509.394,A -85,B 0,C 180,E1 -3907.912,E2 -3907.912} C_VEL
LIN {X 0,Y 537.556,Z 512.738,A -85,B 0,C 180,E1 -3908.869,E2 -3908.869} C_VEL
LIN {X 0,Y 537.506,Z 515.331,A -85,B 0,C 180,E1 -3909.842,E2 -3909.842} C_VEL
LIN {X 0,Y 537.467,Z 517.244,A -85,B 0,C 180,E1 -3910.829,E2 -3910.829} C_VEL
LIN {X 0,Y 537.459,Z 518.477,A -85,B 0,C 180,E1 -3911.827,E2 -3911.827} C_VEL
LIN {X 0,Y 537.446,Z 518.98,A -85,B 0,C 180,E1 -3912.921,E2 -3912.921} C_VEL
LIN {X 0,Y 537.497,Z 518.644,A -85,B 0,C 180,E1 -3914.016,E2 -3914.016} C_VEL
LIN {X 0,Y 537.505,Z 517.507,A -85,B 0,C 180,E1 -3915.085,E2 -3915.085} C_VEL
LIN {X 0,Y 537.502,Z 515.601,A -85,B 0,C 180,E1 -3916.133,E2 -3916.133} C_VEL
LIN {X 0,Y 537.555,Z 512.896,A -85,B 0,C 180,E1 -3917.168,E2 -3917.168} C_VEL
LIN {X 0,Y 537.61,Z 508.37,A -85,B 0,C 180,E1 -3918.437,E2 -3918.437} C_VEL
LIN {X 0,Y 537.657,Z 502.201,A -85,B 0,C 180,E1 -3919.739,E2 -3919.739} C_VEL
LIN {X 0,Y 537.825,Z 494.688,A -85,B 0,C 180,E1 -3920.979,E2 -3920.979} C_VEL
LIN {X 0,Y 538.018,Z 485.89,A -85,B 0,C 180,E1 -3922.124,E2 -3922.124} C_VEL
LIN {X 0,Y 538.187,Z 476.867,A -85,B 0,C 180,E1 -3923.08,E2 -3923.08} C_VEL
LIN {X 0,Y 538.388,Z 467.16,A -85,B 0,C 180,E1 -3923.922,E2 -3923.922} C_VEL
LIN {X 0,Y 538.639,Z 455.421,A -85,B 0,C 180,E1 -3924.735,E2 -3924.735} C_VEL
LIN {X 0,Y 538.845,Z 443.086,A -85,B 0,C 180,E1 -3925.397,E2 -3925.397} C_VEL
LIN {X 0,Y 539.079,Z 431.867,A -85,B 0,C 180,E1 -3925.85,E2 -3925.85} C_VEL
LIN {X 0,Y 539.043,Z 423.895,A -85,B 0,C 180,E1 -3926.098,E2 -3926.098} C_VEL
LIN {X 0,Y 537.543,Z 414.936,A -85,B 0,C 180,E1 -3926.356,E2 -3926.356} C_VEL
LIN {X 0,Y 537.545,Z 410.345,A -85,B 0,C 180,E1 -3929.343,E2 -3929.343} C_VEL
LIN {X 0,Y 537.6,Z 406.46,A -85,B 0,C 180,E1 -3931.925,E2 -3931.925} C_VEL
LIN {X 0,Y 537.651,Z 402.755,A -85,B 0,C 180,E1 -3934.446,E2 -3934.446} C_VEL
LIN {X 0,Y 537.695,Z 399.218,A -85,B 0,C 180,E1 -3936.914,E2 -3936.914} C_VEL
LIN {X 0,Y 537.782,Z 395.636,A -85,B 0,C 180,E1 -3939.338,E2 -3939.338} C_VEL
LIN {X 0,Y 537.843,Z 391.023,A -85,B 0,C 180,E1 -3942.531,E2 -3942.531} C_VEL
LIN {X 0,Y 537.914,Z 386.644,A -85,B 0,C 180,E1 -3945.627,E2 -3945.627} C_VEL
LIN {X 0,Y 537.943,Z 383.481,A -85,B 0,C 180,E1 -3947.934,E2 -3947.934} C_VEL
LIN {X 0,Y 538.043,Z 383.469,A -85,B 0,C 180,E1 -3950.223,E2 -3950.223} C_VEL
LIN {X 0,Y 538.108,Z 383.459,A -85,B 0,C 180,E1 -3953.25,E2 -3953.25} C_VEL
LIN {X 0,Y 538.03,Z 383.47,A -85,B 0,C 180,E1 -3955.505,E2 -3955.505} C_VEL
LIN {X 0,Y 538.162,Z 383.453,A -85,B 0,C 180,E1 -3957.755,E2 -3957.755} C_VEL
LIN {X 0,Y 538.182,Z 383.451,A -85,B 0,C 180,E1 -3960.748,E2 -3960.748} C_VEL
LIN {X 0,Y 538.136,Z 383.455,A -85,B 0,C 180,E1 -3962.995,E2 -3962.995} C_VEL
LIN {X 0,Y 538.123,Z 383.458,A -85,B 0,C 180,E1 -3965.997,E2 -3965.997} C_VEL
LIN {X 0,Y 538.068,Z 383.465,A -85,B 0,C 180,E1 -3969.018,E2 -3969.018} C_VEL
LIN {X 0,Y 538.08,Z 383.463,A -85,B 0,C 180,E1 -3972.063,E2 -3972.063} C_VEL
LIN {X 0,Y 538.042,Z 383.467,A -85,B 0,C 180,E1 -3975.144,E2 -3975.144} C_VEL
LIN {X 0,Y 538.032,Z 383.469,A -85,B 0,C 180,E1 -3978.27,E2 -3978.27} C_VEL
LIN {X 0,Y 538.039,Z 383.467,A -85,B 0,C 180,E1 -3980.651,E2 -3980.651} C_VEL
LIN {X 0,Y 538.021,Z 383.468,A -85,B 0,C 180,E1 -3983.888,E2 -3983.888} C_VEL
LIN {X 0,Y 538.047,Z 383.466,A -85,B 0,C 180,E1 -3986.367,E2 -3986.367} C_VEL
LIN {X 0,Y 538.053,Z 383.466,A -85,B 0,C 180,E1 -3988.939,E2 -3988.939} C_VEL
LIN {X 0,Y 538.012,Z 383.472,A -85,B 0,C 180,E1 -3991.888,E2 -3991.888} C_VEL
LIN {X 0,Y 538.025,Z 383.468,A -85,B 0,C 180,E1 -3994.621,E2 -3994.621} C_VEL
LIN {X 0,Y 538.006,Z 383.473,A -85,B 0,C 180,E1 -3997.171,E2 -3997.171} C_VEL
LIN {X 0,Y 538.053,Z 383.466,A -85,B 0,C 180,E1 -3999.795,E2 -3999.795} C_VEL
LIN {X 0,Y 538.017,Z 383.47,A -85,B 0,C 180,E1 -4002.786,E2 -4002.786} C_VEL
LIN {X 0,Y 538.029,Z 383.468,A -85,B 0,C 180,E1 -4005.141,E2 -4005.141} C_VEL
LIN {X 0,Y 538.04,Z 383.466,A -85,B 0,C 180,E1 -4008.228,E2 -4008.228} C_VEL
LIN {X 0,Y 538.058,Z 383.466,A -85,B 0,C 180,E1 -4010.412,E2 -4010.412} C_VEL
LIN {X 0,Y 538.058,Z 383.471,A -85,B 0,C 180,E1 -4012.502,E2 -4012.502} C_VEL
LIN {X 0,Y 538.672,Z 388.176,A -85,B 0,C 180,E1 -4014.509,E2 -4014.509} C_VEL
LIN {X 0,Y 538.579,Z 393.9,A -85,B 0,C 180,E1 -4016.766,E2 -4016.766} C_VEL
LIN {X 0,Y 538.333,Z 402.136,A -85,B 0,C 180,E1 -4019.877,E2 -4019.877} C_VEL
LIN {X 0,Y 538.193,Z 410.311,A -85,B 0,C 180,E1 -4022.804,E2 -4022.804} C_VEL
LIN {X 0,Y 538.041,Z 418.705,A -85,B 0,C 180,E1 -4025.704,E2 -4025.704} C_VEL
LIN {X 0,Y 537.951,Z 427.069,A -85,B 0,C 180,E1 -4028.543,E2 -4028.543} C_VEL
LIN {X 0,Y 537.85,Z 435.619,A -85,B 0,C 180,E1 -4031.329,E2 -4031.329} C_VEL
LIN {X 0,Y 537.776,Z 444.164,A -85,B 0,C 180,E1 -4034.072,E2 -4034.072} C_VEL
LIN {X 0,Y 537.708,Z 452.192,A -85,B 0,C 180,E1 -4036.658,E2 -4036.658} C_VEL
LIN {X 0,Y 539.252,Z 462.366,A -85,B 0,C 180,E1 -4036.912,E2 -4036.912} C_VEL
LIN {X 0,Y 539.056,Z 474.485,A -85,B 0,C 180,E1 -4037.291,E2 -4037.291} C_VEL
LIN {X 0,Y 538.844,Z 485.497,A -85,B 0,C 180,E1 -4037.764,E2 -4037.764} C_VEL
LIN {X 0,Y 538.645,Z 496.533,A -85,B 0,C 180,E1 -4038.378,E2 -4038.378} C_VEL
LIN {X 0,Y 538.421,Z 507.923,A -85,B 0,C 180,E1 -4039.185,E2 -4039.185} C_VEL
LIN {X 0,Y 538.201,Z 517.602,A -85,B 0,C 180,E1 -4040.037,E2 -4040.037} C_VEL
LIN {X 0,Y 538.015,Z 526.416,A -85,B 0,C 180,E1 -4040.982,E2 -4040.982} C_VEL
LIN {X 0,Y 537.829,Z 535.006,A -85,B 0,C 180,E1 -4042.114,E2 -4042.114} C_VEL
LIN {X 0,Y 537.705,Z 541.87,A -85,B 0,C 180,E1 -4043.245,E2 -4043.245} C_VEL
LIN {X 0,Y 537.676,Z 547.367,A -85,B 0,C 180,E1 -4044.374,E2 -4044.374} C_VEL
LIN {X 0,Y 537.557,Z 551.678,A -85,B 0,C 180,E1 -4045.501,E2 -4045.501} C_VEL
LIN {X 0,Y 537.591,Z 553.959,A -85,B 0,C 180,E1 -4046.252,E2 -4046.252} C_VEL
LIN {X 0,Y 537.551,Z 555.808,A -85,B 0,C 180,E1 -4047.003,E2 -4047.003} C_VEL
LIN {X 0,Y 537.451,Z 558.183,A -85,B 0,C 180,E1 -4048.502,E2 -4048.502} C_VEL
LIN {X 0,Y 537.442,Z 559,A -85,B 0,C 180,E1 -4050,E2 -4050} C_VEL
LIN {X 0,Y 537.451,Z 558.184,A -85,B 0,C 180,E1 -4051.499,E2 -4051.499} C_VEL
LIN {X 0,Y 537.551,Z 555.809,A -85,B 0,C 180,E1 -4052.998,E2 -4052.998} C_VEL
LIN {X 0,Y 537.603,Z 552.895,A -85,B 0,C 180,E1 -4054.123,E2 -4054.123} C_VEL
LIN {X 0,Y 537.587,Z 548.947,A -85,B 0,C 180,E1 -4055.251,E2 -4055.251} C_VEL
LIN {X 0,Y 537.65,Z 544.081,A -85,B 0,C 180,E1 -4056.335,E2 -4056.335} C_VEL
LIN {X 0,Y 537.791,Z 537.465,A -85,B 0,C 180,E1 -4057.509,E2 -4057.509} C_VEL
LIN {X 0,Y 537.973,Z 529.475,A -85,B 0,C 180,E1 -4058.641,E2 -4058.641} C_VEL
LIN {X 0,Y 538.119,Z 521.331,A -85,B 0,C 180,E1 -4059.586,E2 -4059.586} C_VEL
LIN {X 0,Y 538.348,Z 511.395,A -85,B 0,C 180,E1 -4060.531,E2 -4060.531} C_VEL
LIN {X 0,Y 538.556,Z 501.588,A -85,B 0,C 180,E1 -4061.288,E2 -4061.288} C_VEL
LIN {X 0,Y 538.738,Z 490.617,A -85,B 0,C 180,E1 -4061.969,E2 -4061.969} C_VEL
LIN {X 0,Y 538.963,Z 478.097,A -85,B 0,C 180,E1 -4062.568,E2 -4062.568} C_VEL
LIN {X 0,Y 539.208,Z 465.079,A -85,B 0,C 180,E1 -4063.017,E2 -4063.017} C_VEL
LIN {X 0,Y 539.001,Z 460.025,A -85,B 0,C 180,E1 -4063.154,E2 -4063.154} C_VEL
LIN {X 0,Y 537.711,Z 452.19,A -85,B 0,C 180,E1 -4063.343,E2 -4063.343} C_VEL
LIN {X 0,Y 537.777,Z 444.192,A -85,B 0,C 180,E1 -4065.929,E2 -4065.929} C_VEL
LIN {X 0,Y 537.88,Z 435.724,A -85,B 0,C 180,E1 -4068.67,E2 -4068.67} C_VEL
LIN {X 0,Y 537.968,Z 427.224,A -85,B 0,C 180,E1 -4071.456,E2 -4071.456} C_VEL
LIN {X 0,Y 538.089,Z 418.919,A -85,B 0,C 180,E1 -4074.294,E2 -4074.294} C_VEL
LIN {X 0,Y 538.267,Z 410.074,A -85,B 0,C 180,E1 -4077.394,E2 -4077.394} C_VEL
LIN {X 0,Y 538.418,Z 401.11,A -85,B 0,C 180,E1 -4080.602,E2 -4080.602} C_VEL
LIN {X 0,Y 538.618,Z 393.73,A -85,B 0,C 180,E1 -4083.375,E2 -4083.375} C_VEL
LIN {X 0,Y 538.703,Z 388.289,A -85,B 0,C 180,E1 -4085.489,E2 -4085.489} C_VEL
LIN {X 0,Y 538.059,Z 383.465,A -85,B 0,C 180,E1 -4087.498,E2 -4087.498} C_VEL
LIN {X 0,Y 538.051,Z 383.465,A -85,B 0,C 180,E1 -4090.776,E2 -4090.776} C_VEL
LIN {X 0,Y 538.005,Z 383.471,A -85,B 0,C 180,E1 -4093.816,E2 -4093.816} C_VEL
LIN {X 0,Y 538.028,Z 383.469,A -85,B 0,C 180,E1 -4097.012,E2 -4097.012} C_VEL
LIN {X 0,Y 538.049,Z 383.466,A -85,B 0,C 180,E1 -4099.253,E2 -4099.253} C_VEL
LIN {X 0,Y 537.994,Z 383.472,A -85,B 0,C 180,E1 -4102.122,E2 -4102.122} C_VEL
LIN {X 0,Y 538.008,Z 383.47,A -85,B 0,C 180,E1 -4104.916,E2 -4104.916} C_VEL
LIN {X 0,Y 538.018,Z 383.47,A -85,B 0,C 180,E1 -4107.617,E2 -4107.617} C_VEL
LIN {X 0,Y 538.018,Z 383.47,A -85,B 0,C 180,E1 -4110.239,E2 -4110.239} C_VEL
LIN {X 0,Y 538.058,Z 383.465,A -85,B 0,C 180,E1 -4112.796,E2 -4112.796} C_VEL
LIN {X 0,Y 538.049,Z 383.465,A -85,B 0,C 180,E1 -4115.292,E2 -4115.292} C_VEL
LIN {X 0,Y 538.023,Z 383.469,A -85,B 0,C 180,E1 -4118.546,E2 -4118.546} C_VEL
LIN {X 0,Y 538.034,Z 383.469,A -85,B 0,C 180,E1 -4120.94,E2 -4120.94} C_VEL
LIN {X 0,Y 538.025,Z 383.471,A -85,B 0,C 180,E1 -4123.299,E2 -4123.299} C_VEL
LIN {X 0,Y 538.064,Z 383.465,A -85,B 0,C 180,E1 -4125.631,E2 -4125.631} C_VEL
LIN {X 0,Y 538.077,Z 383.461,A -85,B 0,C 180,E1 -4128.701,E2 -4128.701} C_VEL
LIN {X 0,Y 538.087,Z 383.461,A -85,B 0,C 180,E1 -4131.74,E2 -4131.74} C_VEL
LIN {X 0,Y 538.162,Z 383.45,A -85,B 0,C 180,E1 -4134.755,E2 -4134.755} C_VEL
LIN {X 0,Y 538.164,Z 383.451,A -85,B 0,C 180,E1 -4137.755,E2 -4137.755} C_VEL
LIN {X 0,Y 538.183,Z 383.448,A -85,B 0,C 180,E1 -4140.748,E2 -4140.748} C_VEL
LIN {X 0,Y 538.141,Z 383.453,A -85,B 0,C 180,E1 -4142.994,E2 -4142.994} C_VEL
LIN {X 0,Y 538.124,Z 383.457,A -85,B 0,C 180,E1 -4145.997,E2 -4145.997} C_VEL
LIN {X 0,Y 538.071,Z 383.462,A -85,B 0,C 180,E1 -4149.018,E2 -4149.018} C_VEL
LIN {X 0,Y 538.083,Z 383.462,A -85,B 0,C 180,E1 -4152.062,E2 -4152.062} C_VEL
LIN {X 0,Y 538.045,Z 383.465,A -85,B 0,C 180,E1 -4155.144,E2 -4155.144} C_VEL
LIN {X 0,Y 538.032,Z 383.467,A -85,B 0,C 180,E1 -4158.27,E2 -4158.27} C_VEL
LIN {X 0,Y 538.038,Z 383.467,A -85,B 0,C 180,E1 -4160.651,E2 -4160.651} C_VEL
LIN {X 0,Y 538.005,Z 383.472,A -85,B 0,C 180,E1 -4163.888,E2 -4163.888} C_VEL
LIN {X 0,Y 538.041,Z 383.468,A -85,B 0,C 180,E1 -4166.367,E2 -4166.367} C_VEL
LIN {X 0,Y 538.03,Z 383.468,A -85,B 0,C 180,E1 -4168.933,E2 -4168.933} C_VEL
LIN {X 0,Y 538.015,Z 383.468,A -85,B 0,C 180,E1 -4171.888,E2 -4171.888} C_VEL
LIN {X 0,Y 538.028,Z 383.47,A -85,B 0,C 180,E1 -4174.62,E2 -4174.62} C_VEL
LIN {X 0,Y 538.009,Z 383.47,A -85,B 0,C 180,E1 -4177.171,E2 -4177.171} C_VEL
LIN {X 0,Y 538.017,Z 383.467,A -85,B 0,C 180,E1 -4180.258,E2 -4180.258} C_VEL
LIN {X 0,Y 537.369,Z 383.551,A -85,B 0,C 180,E1 -4180.883,E2 -4180.883} C_VEL
LIN {X 0,Y 534.524,Z 383.906,A -85,B 0,C 180,E1 -4181.898,E2 -4181.898} C_VEL
LIN {X 0,Y 532.101,Z 384.207,A -85,B 0,C 180,E1 -4182.716,E2 -4182.716} C_VEL
LIN {X 0,Y 531.052,Z 384.336,A -85,B 0,C 180,E1 -4183.347,E2 -4183.347} C_VEL
LIN {X 0,Y 530.962,Z 384.346,A -85,B 0,C 180,E1 -4183.56,E2 -4183.56} C_VEL
LIN {X 0,Y 530.956,Z 384.35,A -85,B 0,C 180,E1 -4186.504,E2 -4186.504} C_VEL
LIN {X 0,Y 530.99,Z 384.346,A -85,B 0,C 180,E1 -4188.976,E2 -4188.976} C_VEL
LIN {X 0,Y 530.957,Z 384.349,A -85,B 0,C 180,E1 -4191.529,E2 -4191.529} C_VEL
LIN {X 0,Y 530.978,Z 384.345,A -85,B 0,C 180,E1 -4194.382,E2 -4194.382} C_VEL
LIN {X 0,Y 530.969,Z 384.348,A -85,B 0,C 180,E1 -4197.133,E2 -4197.133} C_VEL
LIN {X 0,Y 530.972,Z 384.348,A -85,B 0,C 180,E1 -4199.803,E2 -4199.803} C_VEL
LIN {X 0,Y 531.014,Z 384.341,A -85,B 0,C 180,E1 -4202.468,E2 -4202.468} C_VEL
LIN {X 0,Y 531.008,Z 384.341,A -85,B 0,C 180,E1 -4204.942,E2 -4204.942} C_VEL
LIN {X 0,Y 530.974,Z 384.347,A -85,B 0,C 180,E1 -4208.247,E2 -4208.247} C_VEL
LIN {X 0,Y 530.996,Z 384.344,A -85,B 0,C 180,E1 -4210.677,E2 -4210.677} C_VEL
LIN {X 0,Y 530.983,Z 384.344,A -85,B 0,C 180,E1 -4213.071,E2 -4213.071} C_VEL
LIN {X 0,Y 531.022,Z 384.341,A -85,B 0,C 180,E1 -4215.436,E2 -4215.436} C_VEL
LIN {X 0,Y 531.04,Z 384.339,A -85,B 0,C 180,E1 -4218.55,E2 -4218.55} C_VEL
LIN {X 0,Y 531.055,Z 384.335,A -85,B 0,C 180,E1 -4221.629,E2 -4221.629} C_VEL
LIN {X 0,Y 531.122,Z 384.33,A -85,B 0,C 180,E1 -4224.685,E2 -4224.685} C_VEL
LIN {X 0,Y 531.143,Z 384.324,A -85,B 0,C 180,E1 -4227.725,E2 -4227.725} C_VEL
LIN {X 0,Y 531.155,Z 384.325,A -85,B 0,C 180,E1 -4230.758,E2 -4230.758} C_VEL
LIN {X 0,Y 531.106,Z 384.331,A -85,B 0,C 180,E1 -4233.034,E2 -4233.034} C_VEL
LIN {X 0,Y 531.073,Z 384.334,A -85,B 0,C 180,E1 -4236.077,E2 -4236.077} C_VEL
LIN {X 0,Y 530.899,Z 384.358,A -85,B 0,C 180,E1 -4238.373,E2 -4238.373} C_VEL
LIN {X 0,Y 530.82,Z 387.316,A -85,B 0,C 180,E1 -4240.682,E2 -4240.682} C_VEL
LIN {X 0,Y 530.71,Z 391.754,A -85,B 0,C 180,E1 -4243.79,E2 -4243.79} C_VEL
LIN {X 0,Y 530.646,Z 395.166,A -85,B 0,C 180,E1 -4246.148,E2 -4246.148} C_VEL
LIN {X 0,Y 530.577,Z 398.663,A -85,B 0,C 180,E1 -4248.536,E2 -4248.536} C_VEL
LIN {X 0,Y 530.502,Z 402.238,A -85,B 0,C 180,E1 -4250.958,E2 -4250.958} C_VEL
LIN {X 0,Y 530.501,Z 406.59,A -85,B 0,C 180,E1 -4253.921,E2 -4253.921} C_VEL
LIN {X 0,Y 530.408,Z 410.87,A -85,B 0,C 180,E1 -4256.776,E2 -4256.776} C_VEL
LIN {X 0,Y 530.419,Z 415.123,A -85,B 0,C 180,E1 -4259.547,E2 -4259.547} C_VEL
LIN {X 0,Y 532.285,Z 427,A -85,B 0,C 180,E1 -4259.909,E2 -4259.909} C_VEL
LIN {X 0,Y 532.022,Z 440.18,A -85,B 0,C 180,E1 -4260.393,E2 -4260.393} C_VEL
LIN {X 0,Y 531.746,Z 451.391,A -85,B 0,C 180,E1 -4260.952,E2 -4260.952} C_VEL
LIN {X 0,Y 531.442,Z 463.159,A -85,B 0,C 180,E1 -4261.713,E2 -4261.713} C_VEL
LIN {X 0,Y 531.278,Z 474.419,A -85,B 0,C 180,E1 -4262.641,E2 -4262.641} C_VEL
LIN {X 0,Y 531.031,Z 483.888,A -85,B 0,C 180,E1 -4263.608,E2 -4263.608} C_VEL
LIN {X 0,Y 530.77,Z 493.392,A -85,B 0,C 180,E1 -4264.82,E2 -4264.82} C_VEL
LIN {X 0,Y 530.68,Z 500.052,A -85,B 0,C 180,E1 -4265.871,E2 -4265.871} C_VEL
LIN {X 0,Y 530.566,Z 505.72,A -85,B 0,C 180,E1 -4266.971,E2 -4266.971} C_VEL
LIN {X 0,Y 530.488,Z 510.08,A -85,B 0,C 180,E1 -4268.027,E2 -4268.027} C_VEL
LIN {X 0,Y 530.432,Z 514.608,A -85,B 0,C 180,E1 -4269.492,E2 -4269.492} C_VEL
LIN {X 0,Y 530.359,Z 517.46,A -85,B 0,C 180,E1 -4270.946,E2 -4270.946} C_VEL
LIN {X 0,Y 530.36,Z 518.895,A -85,B 0,C 180,E1 -4272.517,E2 -4272.517} C_VEL
LIN {X 0,Y 530.352,Z 518.899,A -85,B 0,C 180,E1 -4273.557,E2 -4273.557} C_VEL
LIN {X 0,Y 530.402,Z 518.135,A -85,B 0,C 180,E1 -4274.608,E2 -4274.608} C_VEL
LIN {X 0,Y 530.414,Z 516.575,A -85,B 0,C 180,E1 -4275.683,E2 -4275.683} C_VEL
LIN {X 0,Y 530.448,Z 513.139,A -85,B 0,C 180,E1 -4277.136,E2 -4277.136} C_VEL
LIN {X 0,Y 530.534,Z 508.323,A -85,B 0,C 180,E1 -4278.52,E2 -4278.52} C_VEL
LIN {X 0,Y 530.598,Z 501.899,A -85,B 0,C 180,E1 -4279.886,E2 -4279.886} C_VEL
LIN {X 0,Y 530.746,Z 495.378,A -85,B 0,C 180,E1 -4280.979,E2 -4280.979} C_VEL
LIN {X 0,Y 530.97,Z 486.844,A -85,B 0,C 180,E1 -4282.133,E2 -4282.133} C_VEL
LIN {X 0,Y 531.172,Z 478.016,A -85,B 0,C 180,E1 -4283.104,E2 -4283.104} C_VEL
LIN {X 0,Y 531.388,Z 468.376,A -85,B 0,C 180,E1 -4283.974,E2 -4283.974} C_VEL
LIN {X 0,Y 531.671,Z 457.022,A -85,B 0,C 180,E1 -4284.799,E2 -4284.799} C_VEL
LIN {X 0,Y 531.875,Z 444.678,A -85,B 0,C 180,E1 -4285.491,E2 -4285.491} C_VEL
LIN {X 0,Y 532.183,Z 431.778,A -85,B 0,C 180,E1 -4286.029,E2 -4286.029} C_VEL
LIN {X 0,Y 532.13,Z 424.738,A -85,B 0,C 180,E1 -4286.253,E2 -4286.253} C_VEL
LIN {X 0,Y 530.467,Z 415.157,A -85,B 0,C 180,E1 -4286.535,E2 -4286.535} C_VEL
LIN {X 0,Y 530.462,Z 410.727,A -85,B 0,C 180,E1 -4289.447,E2 -4289.447} C_VEL
LIN {X 0,Y 530.54,Z 406.113,A -85,B 0,C 180,E1 -4292.564,E2 -4292.564} C_VEL
LIN {X 0,Y 530.57,Z 402.715,A -85,B 0,C 180,E1 -4294.92,E2 -4294.92} C_VEL
LIN {X 0,Y 530.644,Z 399.158,A -85,B 0,C 180,E1 -4297.413,E2 -4297.413} C_VEL
LIN {X 0,Y 530.757,Z 395.304,A -85,B 0,C 180,E1 -4300.074,E2 -4300.074} C_VEL
LIN {X 0,Y 530.784,Z 391.072,A -85,B 0,C 180,E1 -4303.064,E2 -4303.064} C_VEL
LIN {X 0,Y 530.849,Z 387.725,A -85,B 0,C 180,E1 -4305.431,E2 -4305.431} C_VEL
LIN {X 0,Y 530.868,Z 384.46,A -85,B 0,C 180,E1 -4307.771,E2 -4307.771} C_VEL
LIN {X 0,Y 530.992,Z 384.347,A -85,B 0,C 180,E1 -4310.092,E2 -4310.092} C_VEL
LIN {X 0,Y 531.078,Z 384.334,A -85,B 0,C 180,E1 -4312.977,E2 -4312.977} C_VEL
LIN {X 0,Y 531.12,Z 384.33,A -85,B 0,C 180,E1 -4314.685,E2 -4314.685} C_VEL
LIN {X 0,Y 531.135,Z 384.329,A -85,B 0,C 180,E1 -4317.725,E2 -4317.725} C_VEL
LIN {X 0,Y 531.152,Z 384.326,A -85,B 0,C 180,E1 -4320.758,E2 -4320.758} C_VEL
LIN {X 0,Y 531.102,Z 384.331,A -85,B 0,C 180,E1 -4323.034,E2 -4323.034} C_VEL
LIN {X 0,Y 531.082,Z 384.334,A -85,B 0,C 180,E1 -4326.077,E2 -4326.077} C_VEL
LIN {X 0,Y 531.028,Z 384.341,A -85,B 0,C 180,E1 -4329.138,E2 -4329.138} C_VEL
LIN {X 0,Y 531.037,Z 384.341,A -85,B 0,C 180,E1 -4332.225,E2 -4332.225} C_VEL
LIN {X 0,Y 530.993,Z 384.346,A -85,B 0,C 180,E1 -4335.35,E2 -4335.35} C_VEL
LIN {X 0,Y 531.013,Z 384.342,A -85,B 0,C 180,E1 -4337.723,E2 -4337.723} C_VEL
LIN {X 0,Y 530.999,Z 384.343,A -85,B 0,C 180,E1 -4340.938,E2 -4340.938} C_VEL
LIN {X 0,Y 530.977,Z 384.345,A -85,B 0,C 180,E1 -4344.225,E2 -4344.225} C_VEL
LIN {X 0,Y 531.009,Z 384.344,A -85,B 0,C 180,E1 -4346.744,E2 -4346.744} C_VEL
LIN {X 0,Y 530.998,Z 384.343,A -85,B 0,C 180,E1 -4349.322,E2 -4349.322} C_VEL
LIN {X 0,Y 530.968,Z 384.349,A -85,B 0,C 180,E1 -4352.102,E2 -4352.102} C_VEL
LIN {X 0,Y 530.982,Z 384.347,A -85,B 0,C 180,E1 -4354.854,E2 -4354.854} C_VEL
LIN {X 0,Y 530.965,Z 384.349,A -85,B 0,C 180,E1 -4357.508,E2 -4357.508} C_VEL
LIN {X 0,Y 531.025,Z 384.342,A -85,B 0,C 180,E1 -4360.429,E2 -4360.429} C_VEL
LIN {X 0,Y 530.963,Z 384.35,A -85,B 0,C 180,E1 -4363.495,E2 -4363.495} C_VEL
LIN {X 0,Y 530.953,Z 384.351,A -85,B 0,C 180,E1 -4366.505,E2 -4366.505} C_VEL
LIN {X 0,Y 531.026,Z 384.342,A -85,B 0,C 180,E1 -4369.572,E2 -4369.572} C_VEL
LIN {X 0,Y 531.035,Z 384.547,A -85,B 0,C 180,E1 -4372.379,E2 -4372.379} C_VEL
LIN {X 0,Y 531.564,Z 387.673,A -85,B 0,C 180,E1 -4373.756,E2 -4373.756} C_VEL
LIN {X 0,Y 531.674,Z 392.691,A -85,B 0,C 180,E1 -4375.821,E2 -4375.821} C_VEL
LIN {X 0,Y 531.424,Z 399.628,A -85,B 0,C 180,E1 -4378.508,E2 -4378.508} C_VEL
LIN {X 0,Y 531.239,Z 406.742,A -85,B 0,C 180,E1 -4381.191,E2 -4381.191} C_VEL
LIN {X 0,Y 531.065,Z 415.026,A -85,B 0,C 180,E1 -4384.145,E2 -4384.145} C_VEL
LIN {X 0,Y 530.957,Z 423.298,A -85,B 0,C 180,E1 -4387.016,E2 -4387.016} C_VEL
LIN {X 0,Y 530.847,Z 432.243,A -85,B 0,C 180,E1 -4390.05,E2 -4390.05} C_VEL
LIN {X 0,Y 530.756,Z 441.474,A -85,B 0,C 180,E1 -4393.064,E2 -4393.064} C_VEL
LIN {X 0,Y 530.647,Z 449.989,A -85,B 0,C 180,E1 -4395.818,E2 -4395.818} C_VEL
LIN {X 0,Y 530.636,Z 452.036,A -85,B 0,C 180,E1 -4396.477,E2 -4396.477} C_VEL
LIN {X 0,Y 532.308,Z 463.154,A -85,B 0,C 180,E1 -4396.763,E2 -4396.763} C_VEL
LIN {X 0,Y 532.11,Z 475.694,A -85,B 0,C 180,E1 -4397.171,E2 -4397.171} C_VEL
LIN {X 0,Y 531.861,Z 487.367,A -85,B 0,C 180,E1 -4397.698,E2 -4397.698} C_VEL
LIN {X 0,Y 531.645,Z 498.383,A -85,B 0,C 180,E1 -4398.345,E2 -4398.345} C_VEL
LIN {X 0,Y 531.407,Z 509.095,A -85,B 0,C 180,E1 -4399.137,E2 -4399.137} C_VEL
LIN {X 0,Y 531.114,Z 519.543,A -85,B 0,C 180,E1 -4400.095,E2 -4400.095} C_VEL
LIN {X 0,Y 530.931,Z 527.995,A -85,B 0,C 180,E1 -4401.052,E2 -4401.052} C_VEL
LIN {X 0,Y 530.758,Z 536.237,A -85,B 0,C 180,E1 -4402.2,E2 -4402.2} C_VEL
LIN {X 0,Y 530.598,Z 543.269,A -85,B 0,C 180,E1 -4403.419,E2 -4403.419} C_VEL
LIN {X 0,Y 530.524,Z 548.951,A -85,B 0,C 180,E1 -4404.68,E2 -4404.68} C_VEL
LIN {X 0,Y 530.522,Z 552.895,A -85,B 0,C 180,E1 -4405.822,E2 -4405.822} C_VEL
LIN {X 0,Y 530.457,Z 555.807,A -85,B 0,C 180,E1 -4406.962,E2 -4406.962} C_VEL
LIN {X 0,Y 530.411,Z 557.194,A -85,B 0,C 180,E1 -4407.722,E2 -4407.722} C_VEL
LIN {X 0,Y 530.344,Z 558.786,A -85,B 0,C 180,E1 -4409.241,E2 -4409.241} C_VEL
LIN {X 0,Y 530.342,Z 559,A -85,B 0,C 180,E1 -4410,E2 -4410} C_VEL
LIN {X 0,Y 530.361,Z 558.183,A -85,B 0,C 180,E1 -4411.519,E2 -4411.519} C_VEL
LIN {X 0,Y 530.411,Z 557.196,A -85,B 0,C 180,E1 -4412.278,E2 -4412.278} C_VEL
LIN {X 0,Y 530.457,Z 555.809,A -85,B 0,C 180,E1 -4413.038,E2 -4413.038} C_VEL
LIN {X 0,Y 530.523,Z 552.894,A -85,B 0,C 180,E1 -4414.179,E2 -4414.179} C_VEL
LIN {X 0,Y 530.524,Z 548.947,A -85,B 0,C 180,E1 -4415.321,E2 -4415.321} C_VEL
LIN {X 0,Y 530.599,Z 543.262,A -85,B 0,C 180,E1 -4416.582,E2 -4416.582} C_VEL
LIN {X 0,Y 530.758,Z 536.234,A -85,B 0,C 180,E1 -4417.801,E2 -4417.801} C_VEL
LIN {X 0,Y 530.931,Z 527.99,A -85,B 0,C 180,E1 -4418.948,E2 -4418.948} C_VEL
LIN {X 0,Y 531.114,Z 519.538,A -85,B 0,C 180,E1 -4419.906,E2 -4419.906} C_VEL
LIN {X 0,Y 531.41,Z 509.088,A -85,B 0,C 180,E1 -4420.863,E2 -4420.863} C_VEL
LIN {X 0,Y 531.634,Z 497.34,A -85,B 0,C 180,E1 -4421.726,E2 -4421.726} C_VEL
LIN {X 0,Y 531.9,Z 485.432,A -85,B 0,C 180,E1 -4422.399,E2 -4422.399} C_VEL
LIN {X 0,Y 532.157,Z 473.07,A -85,B 0,C 180,E1 -4422.926,E2 -4422.926} C_VEL
LIN {X 0,Y 532.136,Z 461.295,A -85,B 0,C 180,E1 -4423.291,E2 -4423.291} C_VEL
LIN {X 0,Y 530.634,Z 452.076,A -85,B 0,C 180,E1 -4423.524,E2 -4423.524} C_VEL
LIN {X 0,Y 530.712,Z 442.804,A -85,B 0,C 180,E1 -4426.542,E2 -4426.542} C_VEL
LIN {X 0,Y 530.837,Z 434.329,A -85,B 0,C 180,E1 -4429.329,E2 -4429.329} C_VEL
LIN {X 0,Y 530.953,Z 426.051,A -85,B 0,C 180,E1 -4432.095,E2 -4432.095} C_VEL
LIN {X 0,Y 531.062,Z 417.596,A -85,B 0,C 180,E1 -4435.055,E2 -4435.055} C_VEL
LIN {X 0,Y 531.221,Z 409.312,A -85,B 0,C 180,E1 -4438.012,E2 -4438.012} C_VEL
LIN {X 0,Y 531.408,Z 401.907,A -85,B 0,C 180,E1 -4440.723,E2 -4440.723} C_VEL
LIN {X 0,Y 531.631,Z 394.038,A -85,B 0,C 180,E1 -4443.726,E2 -4443.726} C_VEL
LIN {X 0,Y 531.724,Z 389.394,A -85,B 0,C 180,E1 -4445.561,E2 -4445.561} C_VEL
LIN {X 0,Y 531.015,Z 384.342,A -85,B 0,C 180,E1 -4447.683,E2 -4447.683} C_VEL
LIN {X 0,Y 530.984,Z 384.345,A -85,B 0,C 180,E1 -4450.433,E2 -4450.433} C_VEL
LIN {X 0,Y 530.963,Z 384.349,A -85,B 0,C 180,E1 -4453.281,E2 -4453.281} C_VEL
LIN {X 0,Y 530.979,Z 384.346,A -85,B 0,C 180,E1 -4455.622,E2 -4455.622} C_VEL
LIN {X 0,Y 530.994,Z 384.344,A -85,B 0,C 180,E1 -4458.564,E2 -4458.564} C_VEL
LIN {X 0,Y 530.958,Z 384.349,A -85,B 0,C 180,E1 -4461.529,E2 -4461.529} C_VEL
LIN {X 0,Y 530.976,Z 384.347,A -85,B 0,C 180,E1 -4464.381,E2 -4464.381} C_VEL
LIN {X 0,Y 530.967,Z 384.347,A -85,B 0,C 180,E1 -4467.133,E2 -4467.133} C_VEL
LIN {X 0,Y 530.97,Z 384.346,A -85,B 0,C 180,E1 -4469.803,E2 -4469.803} C_VEL
LIN {X 0,Y 531.013,Z 384.342,A -85,B 0,C 180,E1 -4472.467,E2 -4472.467} C_VEL
LIN {X 0,Y 531.006,Z 384.344,A -85,B 0,C 180,E1 -4474.942,E2 -4474.942} C_VEL
LIN {X 0,Y 530.972,Z 384.346,A -85,B 0,C 180,E1 -4478.247,E2 -4478.247} C_VEL
LIN {X 0,Y 530.993,Z 384.344,A -85,B 0,C 180,E1 -4480.677,E2 -4480.677} C_VEL
LIN {X 0,Y 530.986,Z 384.345,A -85,B 0,C 180,E1 -4483.071,E2 -4483.071} C_VEL
LIN {X 0,Y 531.019,Z 384.341,A -85,B 0,C 180,E1 -4485.436,E2 -4485.436} C_VEL
LIN {X 0,Y 531.037,Z 384.338,A -85,B 0,C 180,E1 -4488.55,E2 -4488.55} C_VEL
LIN {X 0,Y 531.057,Z 384.337,A -85,B 0,C 180,E1 -4491.629,E2 -4491.629} C_VEL
LIN {X 0,Y 531.121,Z 384.327,A -85,B 0,C 180,E1 -4494.685,E2 -4494.685} C_VEL
LIN {X 0,Y 531.136,Z 384.327,A -85,B 0,C 180,E1 -4497.725,E2 -4497.725} C_VEL
LIN {X 0,Y 531.153,Z 384.324,A -85,B 0,C 180,E1 -4500.758,E2 -4500.758} C_VEL
LIN {X 0,Y 531.107,Z 384.329,A -85,B 0,C 180,E1 -4503.034,E2 -4503.034} C_VEL
LIN {X 0,Y 531.084,Z 384.334,A -85,B 0,C 180,E1 -4506.077,E2 -4506.077} C_VEL
LIN {X 0,Y 531.031,Z 384.339,A -85,B 0,C 180,E1 -4509.138,E2 -4509.138} C_VEL
LIN {X 0,Y 531.041,Z 384.339,A -85,B 0,C 180,E1 -4512.225,E2 -4512.225} C_VEL
LIN {X 0,Y 530.996,Z 384.345,A -85,B 0,C 180,E1 -4515.35,E2 -4515.35} C_VEL
LIN {X 0,Y 530.991,Z 384.344,A -85,B 0,C 180,E1 -4518.521,E2 -4518.521} C_VEL
LIN {X 0,Y 530.999,Z 384.343,A -85,B 0,C 180,E1 -4520.938,E2 -4520.938} C_VEL
LIN {X 0,Y 530.972,Z 384.347,A -85,B 0,C 180,E1 -4524.225,E2 -4524.225} C_VEL
LIN {X 0,Y 531.004,Z 384.342,A -85,B 0,C 180,E1 -4526.744,E2 -4526.744} C_VEL
LIN {X 0,Y 530.981,Z 384.345,A -85,B 0,C 180,E1 -4529.323,E2 -4529.323} C_VEL
LIN {X 0,Y 530.971,Z 384.347,A -85,B 0,C 180,E1 -4532.101,E2 -4532.101} C_VEL
LIN {X 0,Y 530.985,Z 384.346,A -85,B 0,C 180,E1 -4534.853,E2 -4534.853} C_VEL
LIN {X 0,Y 530.967,Z 384.345,A -85,B 0,C 180,E1 -4537.508,E2 -4537.508} C_VEL
LIN {X 0,Y 530.981,Z 384.346,A -85,B 0,C 180,E1 -4540.433,E2 -4540.433} C_VEL
LIN {X 0,Y 530.965,Z 384.346,A -85,B 0,C 180,E1 -4543.495,E2 -4543.495} C_VEL
LIN {X 0,Y 530.962,Z 384.346,A -85,B 0,C 180,E1 -4543.56,E2 -4543.56} C_VEL
LIN {X 0,Y 530.286,Z 384.434,A -85,B 0,C 180,E1 -4544.194,E2 -4544.194} C_VEL
LIN {X 0,Y 527.434,Z 384.789,A -85,B 0,C 180,E1 -4545.222,E2 -4545.222} C_VEL
LIN {X 0,Y 525.031,Z 385.089,A -85,B 0,C 180,E1 -4546.051,E2 -4546.051} C_VEL
LIN {X 0,Y 524,Z 385.216,A -85,B 0,C 180,E1 -4546.69,E2 -4546.69} C_VEL
LIN {X 0,Y 523.917,Z 385.225,A -85,B 0,C 180,E1 -4546.907,E2 -4546.907} C_VEL
LIN {X 0,Y 523.945,Z 385.224,A -85,B 0,C 180,E1 -4548.908,E2 -4548.908} C_VEL
LIN {X 0,Y 523.916,Z 385.224,A -85,B 0,C 180,E1 -4551.898,E2 -4551.898} C_VEL
LIN {X 0,Y 523.936,Z 385.224,A -85,B 0,C 180,E1 -4554.91,E2 -4554.91} C_VEL
LIN {X 0,Y 523.937,Z 385.222,A -85,B 0,C 180,E1 -4557.68,E2 -4557.68} C_VEL
LIN {X 0,Y 523.956,Z 385.222,A -85,B 0,C 180,E1 -4560.677,E2 -4560.677} C_VEL
LIN {X 0,Y 523.976,Z 385.217,A -85,B 0,C 180,E1 -4563.729,E2 -4563.729} C_VEL
LIN {X 0,Y 523.929,Z 385.224,A -85,B 0,C 180,E1 -4566.27,E2 -4566.27} C_VEL
LIN {X 0,Y 523.948,Z 385.221,A -85,B 0,C 180,E1 -4568.767,E2 -4568.767} C_VEL
LIN {X 0,Y 523.952,Z 385.22,A -85,B 0,C 180,E1 -4571.221,E2 -4571.221} C_VEL
LIN {X 0,Y 523.934,Z 385.222,A -85,B 0,C 180,E1 -4573.639,E2 -4573.639} C_VEL
LIN {X 0,Y 523.942,Z 385.222,A -85,B 0,C 180,E1 -4576.028,E2 -4576.028} C_VEL
LIN {X 0,Y 524.015,Z 385.213,A -85,B 0,C 180,E1 -4578.394,E2 -4578.394} C_VEL
LIN {X 0,Y 524.003,Z 385.214,A -85,B 0,C 180,E1 -4581.516,E2 -4581.516} C_VEL
LIN {X 0,Y 524.084,Z 385.206,A -85,B 0,C 180,E1 -4584.613,E2 -4584.613} C_VEL
LIN {X 0,Y 524.115,Z 385.2,A -85,B 0,C 180,E1 -4587.694,E2 -4587.694} C_VEL
LIN {X 0,Y 524.125,Z 385.2,A -85,B 0,C 180,E1 -4590.768,E2 -4590.768} C_VEL
LIN {X 0,Y 524.073,Z 385.207,A -85,B 0,C 180,E1 -4593.075,E2 -4593.075} C_VEL
LIN {X 0,Y 524.031,Z 385.211,A -85,B 0,C 180,E1 -4596.159,E2 -4596.159} C_VEL
LIN {X 0,Y 523.834,Z 385.238,A -85,B 0,C 180,E1 -4598.486,E2 -4598.486} C_VEL
LIN {X 0,Y 523.747,Z 389.384,A -85,B 0,C 180,E1 -4601.611,E2 -4601.611} C_VEL
LIN {X 0,Y 523.647,Z 394.068,A -85,B 0,C 180,E1 -4604.91,E2 -4604.91} C_VEL
LIN {X 0,Y 523.539,Z 398.529,A -85,B 0,C 180,E1 -4607.984,E2 -4607.984} C_VEL
LIN {X 0,Y 523.465,Z 402.096,A -85,B 0,C 180,E1 -4610.43,E2 -4610.43} C_VEL
LIN {X 0,Y 523.421,Z 405.74,A -85,B 0,C 180,E1 -4612.916,E2 -4612.916} C_VEL
LIN {X 0,Y 523.378,Z 410.136,A -85,B 0,C 180,E1 -4615.883,E2 -4615.883} C_VEL
LIN {X 0,Y 523.324,Z 414.697,A -85,B 0,C 180,E1 -4618.911,E2 -4618.911} C_VEL
LIN {X 0,Y 523.349,Z 415.379,A -85,B 0,C 180,E1 -4619.359,E2 -4619.359} C_VEL
LIN {X 0,Y 525.393,Z 427.628,A -85,B 0,C 180,E1 -4619.748,E2 -4619.748} C_VEL
LIN {X 0,Y 525.107,Z 440.661,A -85,B 0,C 180,E1 -4620.236,E2 -4620.236} C_VEL
LIN {X 0,Y 524.789,Z 451.976,A -85,B 0,C 180,E1 -4620.81,E2 -4620.81} C_VEL
LIN {X 0,Y 524.511,Z 462.632,A -85,B 0,C 180,E1 -4621.504,E2 -4621.504} C_VEL
LIN {X 0,Y 524.264,Z 473.843,A -85,B 0,C 180,E1 -4622.426,E2 -4622.426} C_VEL
LIN {X 0,Y 524.02,Z 483.032,A -85,B 0,C 180,E1 -4623.358,E2 -4623.358} C_VEL
LIN {X 0,Y 523.809,Z 492.035,A -85,B 0,C 180,E1 -4624.485,E2 -4624.485} C_VEL
LIN {X 0,Y 523.602,Z 499.926,A -85,B 0,C 180,E1 -4625.723,E2 -4625.723} C_VEL
LIN {X 0,Y 523.532,Z 505.096,A -85,B 0,C 180,E1 -4626.726,E2 -4626.726} C_VEL
LIN {X 0,Y 523.404,Z 510.863,A -85,B 0,C 180,E1 -4628.145,E2 -4628.145} C_VEL
LIN {X 0,Y 523.34,Z 515.009,A -85,B 0,C 180,E1 -4629.588,E2 -4629.588} C_VEL
LIN {X 0,Y 523.25,Z 517.856,A -85,B 0,C 180,E1 -4631.157,E2 -4631.157} C_VEL
LIN {X 0,Y 523.263,Z 518.887,A -85,B 0,C 180,E1 -4632.378,E2 -4632.378} C_VEL
LIN {X 0,Y 523.25,Z 518.949,A -85,B 0,C 180,E1 -4633.506,E2 -4633.506} C_VEL
LIN {X 0,Y 523.303,Z 518.189,A -85,B 0,C 180,E1 -4634.619,E2 -4634.619} C_VEL
LIN {X 0,Y 523.315,Z 516.658,A -85,B 0,C 180,E1 -4635.705,E2 -4635.705} C_VEL
LIN {X 0,Y 523.374,Z 513.148,A -85,B 0,C 180,E1 -4637.22,E2 -4637.22} C_VEL
LIN {X 0,Y 523.44,Z 509.499,A -85,B 0,C 180,E1 -4638.32,E2 -4638.32} C_VEL
LIN {X 0,Y 523.492,Z 503.882,A -85,B 0,C 180,E1 -4639.626,E2 -4639.626} C_VEL
LIN {X 0,Y 523.676,Z 496.804,A -85,B 0,C 180,E1 -4640.893,E2 -4640.893} C_VEL
LIN {X 0,Y 523.834,Z 489.941,A -85,B 0,C 180,E1 -4641.891,E2 -4641.891} C_VEL
LIN {X 0,Y 524.03,Z 481.729,A -85,B 0,C 180,E1 -4642.878,E2 -4642.878} C_VEL
LIN {X 0,Y 524.317,Z 471.747,A -85,B 0,C 180,E1 -4643.858,E2 -4643.858} C_VEL
LIN {X 0,Y 524.66,Z 460.657,A -85,B 0,C 180,E1 -4644.725,E2 -4644.725} C_VEL
LIN {X 0,Y 524.915,Z 448.16,A -85,B 0,C 180,E1 -4645.492,E2 -4645.492} C_VEL
LIN {X 0,Y 525.205,Z 435.764,A -85,B 0,C 180,E1 -4646.061,E2 -4646.061} C_VEL
LIN {X 0,Y 525.161,Z 425.309,A -85,B 0,C 180,E1 -4646.422,E2 -4646.422} C_VEL
LIN {X 0,Y 523.394,Z 415.475,A -85,B 0,C 180,E1 -4646.711,E2 -4646.711} C_VEL
LIN {X 0,Y 523.379,Z 411.532,A -85,B 0,C 180,E1 -4649.318,E2 -4649.318} C_VEL
LIN {X 0,Y 523.482,Z 407.011,A -85,B 0,C 180,E1 -4652.384,E2 -4652.384} C_VEL
LIN {X 0,Y 523.531,Z 402.7,A -85,B 0,C 180,E1 -4655.408,E2 -4655.408} C_VEL
LIN {X 0,Y 523.615,Z 399.085,A -85,B 0,C 180,E1 -4657.925,E2 -4657.925} C_VEL
LIN {X 0,Y 523.699,Z 395.582,A -85,B 0,C 180,E1 -4660.397,E2 -4660.397} C_VEL
LIN {X 0,Y 523.746,Z 391.083,A -85,B 0,C 180,E1 -4663.633,E2 -4663.633} C_VEL
LIN {X 0,Y 523.777,Z 387.707,A -85,B 0,C 180,E1 -4666.024,E2 -4666.024} C_VEL
LIN {X 0,Y 523.837,Z 385.561,A -85,B 0,C 180,E1 -4667.604,E2 -4667.604} C_VEL
LIN {X 0,Y 523.97,Z 385.221,A -85,B 0,C 180,E1 -4669.177,E2 -4669.177} C_VEL
LIN {X 0,Y 524.025,Z 385.215,A -85,B 0,C 180,E1 -4672.293,E2 -4672.293} C_VEL
LIN {X 0,Y 524.081,Z 385.207,A -85,B 0,C 180,E1 -4674.614,E2 -4674.614} C_VEL
LIN {X 0,Y 524.107,Z 385.204,A -85,B 0,C 180,E1 -4677.695,E2 -4677.695} C_VEL
LIN {X 0,Y 524.122,Z 385.202,A -85,B 0,C 180,E1 -4680.768,E2 -4680.768} C_VEL
LIN {X 0,Y 524.069,Z 385.207,A -85,B 0,C 180,E1 -4683.075,E2 -4683.075} C_VEL
LIN {X 0,Y 524.044,Z 385.211,A -85,B 0,C 180,E1 -4686.159,E2 -4686.159} C_VEL
LIN {X 0,Y 523.996,Z 385.216,A -85,B 0,C 180,E1 -4689.262,E2 -4689.262} C_VEL
LIN {X 0,Y 523.999,Z 385.215,A -85,B 0,C 180,E1 -4691.74,E2 -4691.74} C_VEL
LIN {X 0,Y 523.989,Z 385.217,A -85,B 0,C 180,E1 -4695.053,E2 -4695.053} C_VEL
LIN {X 0,Y 523.961,Z 385.22,A -85,B 0,C 180,E1 -4697.969,E2 -4697.969} C_VEL
LIN {X 0,Y 523.969,Z 385.22,A -85,B 0,C 180,E1 -4700.41,E2 -4700.41} C_VEL
LIN {X 0,Y 523.913,Z 385.226,A -85,B 0,C 180,E1 -4702.894,E2 -4702.894} C_VEL
LIN {X 0,Y 523.952,Z 385.222,A -85,B 0,C 180,E1 -4705.419,E2 -4705.419} C_VEL
LIN {X 0,Y 523.968,Z 385.22,A -85,B 0,C 180,E1 -4707.999,E2 -4707.999} C_VEL
LIN {X 0,Y 523.947,Z 385.224,A -85,B 0,C 180,E1 -4710.856,E2 -4710.856} C_VEL
LIN {X 0,Y 523.958,Z 385.221,A -85,B 0,C 180,E1 -4713.735,E2 -4713.735} C_VEL
LIN {X 0,Y 523.919,Z 385.227,A -85,B 0,C 180,E1 -4716.405,E2 -4716.405} C_VEL
LIN {X 0,Y 523.958,Z 385.223,A -85,B 0,C 180,E1 -4719.082,E2 -4719.082} C_VEL
LIN {X 0,Y 523.955,Z 385.223,A -85,B 0,C 180,E1 -4722.119,E2 -4722.119} C_VEL
LIN {X 0,Y 523.952,Z 385.223,A -85,B 0,C 180,E1 -4725.309,E2 -4725.309} C_VEL
LIN {X 0,Y 523.972,Z 385.218,A -85,B 0,C 180,E1 -4728.688,E2 -4728.688} C_VEL
LIN {X 0,Y 523.925,Z 385.226,A -85,B 0,C 180,E1 -4731.08,E2 -4731.08} C_VEL
LIN {X 0,Y 523.957,Z 385.387,A -85,B 0,C 180,E1 -4732.141,E2 -4732.141} C_VEL
LIN {X 0,Y 524.603,Z 389.28,A -85,B 0,C 180,E1 -4733.882,E2 -4733.882} C_VEL
LIN {X 0,Y 524.625,Z 394.764,A -85,B 0,C 180,E1 -4736.157,E2 -4736.157} C_VEL
LIN {X 0,Y 524.428,Z 400.685,A -85,B 0,C 180,E1 -4738.49,E2 -4738.49} C_VEL
LIN {X 0,Y 524.188,Z 408.82,A -85,B 0,C 180,E1 -4741.579,E2 -4741.579} C_VEL
LIN {X 0,Y 524.002,Z 417.116,A -85,B 0,C 180,E1 -4744.584,E2 -4744.584} C_VEL
LIN {X 0,Y 523.891,Z 426.194,A -85,B 0,C 180,E1 -4747.765,E2 -4747.765} C_VEL
LIN {X 0,Y 523.757,Z 433.88,A -85,B 0,C 180,E1 -4750.4,E2 -4750.4} C_VEL
LIN {X 0,Y 523.664,Z 442.438,A -85,B 0,C 180,E1 -4753.229,E2 -4753.229} C_VEL
LIN {X 0,Y 523.57,Z 451.785,A -85,B 0,C 180,E1 -4756.291,E2 -4756.291} C_VEL
LIN {X 0,Y 525.368,Z 463.717,A -85,B 0,C 180,E1 -4756.609,E2 -4756.609} C_VEL
LIN {X 0,Y 525.145,Z 476.559,A -85,B 0,C 180,E1 -4757.047,E2 -4757.047} C_VEL
LIN {X 0,Y 524.85,Z 488.799,A -85,B 0,C 180,E1 -4757.629,E2 -4757.629} C_VEL
LIN {X 0,Y 524.639,Z 499.881,A -85,B 0,C 180,E1 -4758.312,E2 -4758.312} C_VEL
LIN {X 0,Y 524.365,Z 511.155,A -85,B 0,C 180,E1 -4759.185,E2 -4759.185} C_VEL
LIN {X 0,Y 524.056,Z 521.153,A -85,B 0,C 180,E1 -4760.155,E2 -4760.155} C_VEL
LIN {X 0,Y 523.832,Z 530.851,A -85,B 0,C 180,E1 -4761.319,E2 -4761.319} C_VEL
LIN {X 0,Y 523.633,Z 538.569,A -85,B 0,C 180,E1 -4762.481,E2 -4762.481} C_VEL
LIN {X 0,Y 523.515,Z 545.678,A -85,B 0,C 180,E1 -4763.835,E2 -4763.835} C_VEL
LIN {X 0,Y 523.383,Z 550.374,A -85,B 0,C 180,E1 -4764.993,E2 -4764.993} C_VEL
LIN {X 0,Y 523.443,Z 553.958,A -85,B 0,C 180,E1 -4766.151,E2 -4766.151} C_VEL
LIN {X 0,Y 523.367,Z 555.807,A -85,B 0,C 180,E1 -4766.921,E2 -4766.921} C_VEL
LIN {X 0,Y 523.335,Z 557.193,A -85,B 0,C 180,E1 -4767.691,E2 -4767.691} C_VEL
LIN {X 0,Y 523.25,Z 558.785,A -85,B 0,C 180,E1 -4769.231,E2 -4769.231} C_VEL
LIN {X 0,Y 523.246,Z 559,A -85,B 0,C 180,E1 -4770,E2 -4770} C_VEL
LIN {X 0,Y 523.275,Z 558.183,A -85,B 0,C 180,E1 -4771.54,E2 -4771.54} C_VEL
LIN {X 0,Y 523.335,Z 557.195,A -85,B 0,C 180,E1 -4772.309,E2 -4772.309} C_VEL
LIN {X 0,Y 523.367,Z 555.809,A -85,B 0,C 180,E1 -4773.079,E2 -4773.079} C_VEL
LIN {X 0,Y 523.441,Z 552.894,A -85,B 0,C 180,E1 -4774.235,E2 -4774.235} C_VEL
LIN {X 0,Y 523.464,Z 548.947,A -85,B 0,C 180,E1 -4775.393,E2 -4775.393} C_VEL
LIN {X 0,Y 523.523,Z 543.712,A -85,B 0,C 180,E1 -4776.581,E2 -4776.581} C_VEL
LIN {X 0,Y 523.665,Z 537.404,A -85,B 0,C 180,E1 -4777.713,E2 -4777.713} C_VEL
LIN {X 0,Y 523.849,Z 529.36,A -85,B 0,C 180,E1 -4778.876,E2 -4778.876} C_VEL
LIN {X 0,Y 524.056,Z 521.163,A -85,B 0,C 180,E1 -4779.845,E2 -4779.845} C_VEL
LIN {X 0,Y 524.33,Z 511.169,A -85,B 0,C 180,E1 -4780.816,E2 -4780.816} C_VEL
LIN {X 0,Y 524.629,Z 499.961,A -85,B 0,C 180,E1 -4781.685,E2 -4781.685} C_VEL
LIN {X 0,Y 524.845,Z 488.829,A -85,B 0,C 180,E1 -4782.372,E2 -4782.372} C_VEL
LIN {X 0,Y 525.145,Z 476.588,A -85,B 0,C 180,E1 -4782.954,E2 -4782.954} C_VEL
LIN {X 0,Y 525.393,Z 463.738,A -85,B 0,C 180,E1 -4783.39,E2 -4783.39} C_VEL
LIN {X 0,Y 523.568,Z 451.898,A -85,B 0,C 180,E1 -4783.71,E2 -4783.71} C_VEL
LIN {X 0,Y 523.665,Z 442.624,A -85,B 0,C 180,E1 -4786.771,E2 -4786.771} C_VEL
LIN {X 0,Y 523.784,Z 434.147,A -85,B 0,C 180,E1 -4789.6,E2 -4789.6} C_VEL
LIN {X 0,Y 523.896,Z 426.402,A -85,B 0,C 180,E1 -4792.236,E2 -4792.236} C_VEL
LIN {X 0,Y 524.008,Z 418.638,A -85,B 0,C 180,E1 -4794.991,E2 -4794.991} C_VEL
LIN {X 0,Y 524.175,Z 410.977,A -85,B 0,C 180,E1 -4797.759,E2 -4797.759} C_VEL
LIN {X 0,Y 524.38,Z 403.302,A -85,B 0,C 180,E1 -4800.617,E2 -4800.617} C_VEL
LIN {X 0,Y 524.598,Z 396.283,A -85,B 0,C 180,E1 -4803.317,E2 -4803.317} C_VEL
LIN {X 0,Y 524.742,Z 390.487,A -85,B 0,C 180,E1 -4805.634,E2 -4805.634} C_VEL
LIN {X 0,Y 523.952,Z 385.223,A -85,B 0,C 180,E1 -4807.889,E2 -4807.889} C_VEL
LIN {X 0,Y 523.943,Z 385.224,A -85,B 0,C 180,E1 -4811.092,E2 -4811.092} C_VEL
LIN {X 0,Y 523.933,Z 385.223,A -85,B 0,C 180,E1 -4814.229,E2 -4814.229} C_VEL
LIN {X 0,Y 523.918,Z 385.225,A -85,B 0,C 180,E1 -4816.833,E2 -4816.833} C_VEL
LIN {X 0,Y 523.94,Z 385.222,A -85,B 0,C 180,E1 -4818.907,E2 -4818.907} C_VEL
LIN {X 0,Y 523.917,Z 385.226,A -85,B 0,C 180,E1 -4821.898,E2 -4821.898} C_VEL
LIN {X 0,Y 523.931,Z 385.223,A -85,B 0,C 180,E1 -4824.91,E2 -4824.91} C_VEL
LIN {X 0,Y 523.935,Z 385.225,A -85,B 0,C 180,E1 -4827.68,E2 -4827.68} C_VEL
LIN {X 0,Y 523.955,Z 385.22,A -85,B 0,C 180,E1 -4830.676,E2 -4830.676} C_VEL
LIN {X 0,Y 523.974,Z 385.22,A -85,B 0,C 180,E1 -4833.728,E2 -4833.728} C_VEL
LIN {X 0,Y 523.927,Z 385.225,A -85,B 0,C 180,E1 -4836.27,E2 -4836.27} C_VEL
LIN {X 0,Y 523.946,Z 385.223,A -85,B 0,C 180,E1 -4838.767,E2 -4838.767} C_VEL
LIN {X 0,Y 523.95,Z 385.222,A -85,B 0,C 180,E1 -4841.221,E2 -4841.221} C_VEL
LIN {X 0,Y 523.937,Z 385.222,A -85,B 0,C 180,E1 -4843.639,E2 -4843.639} C_VEL
LIN {X 0,Y 523.939,Z 385.222,A -85,B 0,C 180,E1 -4846.028,E2 -4846.028} C_VEL
LIN {X 0,Y 524.013,Z 385.214,A -85,B 0,C 180,E1 -4848.394,E2 -4848.394} C_VEL
LIN {X 0,Y 524.005,Z 385.216,A -85,B 0,C 180,E1 -4851.516,E2 -4851.516} C_VEL
LIN {X 0,Y 524.083,Z 385.204,A -85,B 0,C 180,E1 -4854.614,E2 -4854.614} C_VEL
LIN {X 0,Y 524.109,Z 385.202,A -85,B 0,C 180,E1 -4857.694,E2 -4857.694} C_VEL
LIN {X 0,Y 524.123,Z 385.199,A -85,B 0,C 180,E1 -4860.768,E2 -4860.768} C_VEL
LIN {X 0,Y 524.073,Z 385.206,A -85,B 0,C 180,E1 -4863.075,E2 -4863.075} C_VEL
LIN {X 0,Y 524.046,Z 385.21,A -85,B 0,C 180,E1 -4866.159,E2 -4866.159} C_VEL
LIN {X 0,Y 523.999,Z 385.216,A -85,B 0,C 180,E1 -4869.262,E2 -4869.262} C_VEL
LIN {X 0,Y 524.003,Z 385.215,A -85,B 0,C 180,E1 -4871.739,E2 -4871.739} C_VEL
LIN {X 0,Y 523.993,Z 385.216,A -85,B 0,C 180,E1 -4875.052,E2 -4875.052} C_VEL
LIN {X 0,Y 523.964,Z 385.22,A -85,B 0,C 180,E1 -4877.969,E2 -4877.969} C_VEL
LIN {X 0,Y 523.972,Z 385.221,A -85,B 0,C 180,E1 -4880.41,E2 -4880.41} C_VEL
LIN {X 0,Y 523.911,Z 385.227,A -85,B 0,C 180,E1 -4882.894,E2 -4882.894} C_VEL
LIN {X 0,Y 523.952,Z 385.22,A -85,B 0,C 180,E1 -4885.419,E2 -4885.419} C_VEL
LIN {X 0,Y 523.967,Z 385.218,A -85,B 0,C 180,E1 -4887.999,E2 -4887.999} C_VEL
LIN {X 0,Y 523.945,Z 385.223,A -85,B 0,C 180,E1 -4890.855,E2 -4890.855} C_VEL
LIN {X 0,Y 523.961,Z 385.22,A -85,B 0,C 180,E1 -4893.735,E2 -4893.735} C_VEL
LIN {X 0,Y 523.922,Z 385.224,A -85,B 0,C 180,E1 -4896.404,E2 -4896.404} C_VEL
LIN {X 0,Y 523.92,Z 385.225,A -85,B 0,C 180,E1 -4899.085,E2 -4899.085} C_VEL
LIN {X 0,Y 523.952,Z 385.221,A -85,B 0,C 180,E1 -4902.119,E2 -4902.119} C_VEL
LIN {X 0,Y 523.944,Z 385.223,A -85,B 0,C 180,E1 -4905.31,E2 -4905.31} C_VEL
LIN {X 0,Y 523.917,Z 385.225,A -85,B 0,C 180,E1 -4906.907,E2 -4906.907} C_VEL
LIN {X 0,Y 523.253,Z 385.308,A -85,B 0,C 180,E1 -4907.548,E2 -4907.548} C_VEL
LIN {X 0,Y 520.413,Z 385.665,A -85,B 0,C 180,E1 -4908.59,E2 -4908.59} C_VEL
LIN {X 0,Y 518.008,Z 385.967,A -85,B 0,C 180,E1 -4909.429,E2 -4909.429} C_VEL
LIN {X 0,Y 516.97,Z 386.094,A -85,B 0,C 180,E1 -4910.077,E2 -4910.077} C_VEL
LIN {X 0,Y 516.882,Z 386.103,A -85,B 0,C 180,E1 -4910.296,E2 -4910.296} C_VEL
LIN {X 0,Y 516.885,Z 386.101,A -85,B 0,C 180,E1 -4913.342,E2 -4913.342} C_VEL
LIN {X 0,Y 516.912,Z 386.099,A -85,B 0,C 180,E1 -4916.121,E2 -4916.121} C_VEL
LIN {X 0,Y 516.893,Z 386.1,A -85,B 0,C 180,E1 -4918.936,E2 -4918.936} C_VEL
LIN {X 0,Y 516.92,Z 386.095,A -85,B 0,C 180,E1 -4921.585,E2 -4921.585} C_VEL
LIN {X 0,Y 516.934,Z 386.095,A -85,B 0,C 180,E1 -4924.211,E2 -4924.211} C_VEL
LIN {X 0,Y 516.868,Z 386.106,A -85,B 0,C 180,E1 -4926.776,E2 -4926.776} C_VEL
LIN {X 0,Y 516.942,Z 386.093,A -85,B 0,C 180,E1 -4929.732,E2 -4929.732} C_VEL
LIN {X 0,Y 516.922,Z 386.098,A -85,B 0,C 180,E1 -4932.596,E2 -4932.596} C_VEL
LIN {X 0,Y 516.945,Z 386.095,A -85,B 0,C 180,E1 -4935.03,E2 -4935.03} C_VEL
LIN {X 0,Y 516.969,Z 386.091,A -85,B 0,C 180,E1 -4938.234,E2 -4938.234} C_VEL
LIN {X 0,Y 516.968,Z 386.091,A -85,B 0,C 180,E1 -4941.399,E2 -4941.399} C_VEL
LIN {X 0,Y 517.015,Z 386.086,A -85,B 0,C 180,E1 -4943.757,E2 -4943.757} C_VEL
LIN {X 0,Y 517.087,Z 386.075,A -85,B 0,C 180,E1 -4947.663,E2 -4947.663} C_VEL
LIN {X 0,Y 517.095,Z 386.075,A -85,B 0,C 180,E1 -4950.778,E2 -4950.778} C_VEL
LIN {X 0,Y 517.014,Z 386.086,A -85,B 0,C 180,E1 -4953.117,E2 -4953.117} C_VEL
LIN {X 0,Y 516.993,Z 386.088,A -85,B 0,C 180,E1 -4956.243,E2 -4956.243} C_VEL
LIN {X 0,Y 516.783,Z 386.116,A -85,B 0,C 180,E1 -4958.603,E2 -4958.603} C_VEL
LIN {X 0,Y 516.667,Z 390.359,A -85,B 0,C 180,E1 -4961.773,E2 -4961.773} C_VEL
LIN {X 0,Y 516.587,Z 394.906,A -85,B 0,C 180,E1 -4964.998,E2 -4964.998} C_VEL
LIN {X 0,Y 516.47,Z 399.548,A -85,B 0,C 180,E1 -4968.238,E2 -4968.238} C_VEL
LIN {X 0,Y 516.374,Z 403.161,A -85,B 0,C 180,E1 -4970.724,E2 -4970.724} C_VEL
LIN {X 0,Y 516.352,Z 406.834,A -85,B 0,C 180,E1 -4973.248,E2 -4973.248} C_VEL
